(* Logix 5000 project; controller LeakTestAuto vendor 1 type 14 code 226 rev 37.11; software revision 37.01; part 4 of 12 *)
(* tags used below, declared in another part *)
   DateString : String20;
   DateTimeString : String20;
   I_OP220_N3_CONVEYOR_CLEAT : ALIAS FOR Local:3:I.Pt13.Data;
   I_OP220_N3_CONVEYOR_LOAD : ALIAS FOR Local:3:I.Pt12.Data;
   I_OP220_N3_CONVEYOR_UNLOAD : ALIAS FOR Local:3:I.Pt14.Data;
   I_OP220_N3_DUT_PRE_NEST_0 : ALIAS FOR Local:3:I.Pt00.Data;
   I_OP220_N3_DUT_PRE_NEST_1 : ALIAS FOR Local:3:I.Pt01.Data;
   I_OP220_N3_DUT_PRE_NEST_2 : ALIAS FOR Local:3:I.Pt02.Data;
   I_OP220_N3_NEST1_EXTEND : ALIAS FOR Local:3:I.Pt04.Data;
   I_OP220_N3_NEST1_HOME : ALIAS FOR Local:3:I.Pt03.Data;
   I_OP220_N3_NEST2_EXTEND : ALIAS FOR Local:3:I.Pt06.Data;
   I_OP220_N3_NEST2_HOME : ALIAS FOR Local:3:I.Pt05.Data;
   I_OP220_N3_REJECT_BIN_OK : ALIAS FOR Local:3:I.Pt09.Data;
   IOCounterHasRef : BOOL;
   IOTriggerCounts : UDINT[128];
   LastPLCEdit : String20;
   LastPLCEditHistory : String20[20];
   PLC : AOI_PLC;
   ShiftChange : BOOL;
   ShiftNumber : SINT;
   TimeString : String20;
   TON_PLC_BootUp : TIMER;

        [4].Detailed.element_data[2].Variable_code := 13, [4].Detailed.element_data[2].prec_code := 3, [4].Detailed.element_data[2].Unit_code := 12, [4].Detailed.element_data[2].result_measurement := 5.1366444, [4].Detailed.element_data[3].Variable_code := 75, [4].Detailed.element_data[3].prec_code := 2, [4].Detailed.element_data[3].Unit_code := 60, [4].Detailed.element_data[4].Variable_code := 60, [4].Detailed.element_data[4].prec_code := 2, [4].Detailed.element_data[4].Unit_code := 60, [4].Detailed.element_data[4].result_measurement := -0.06984919, [4].Detailed.element_data[5].Variable_code := 56, [4].Detailed.element_data[5].prec_code := 3, [4].Detailed.element_data[5].Unit_code := 41, [4].Detailed.element_data[5].result_measurement := 0.00021420419, [4].Detailed.element_data[6].Variable_code := 55, [4].Detailed.element_data[6].prec_code := 3, [4].Detailed.element_data[6].Unit_code := 12, [4].Detailed.element_data[6].result_measurement := 5.1366444, [4].Detailed.element_data[7].Variable_code := 58, [4].Detailed.element_data[7].prec_code := 2, [4].Detailed.element_data[7].Unit_code := 60, [4].Detailed.element_data[7].result_measurement := -1.0002404, [4].Detailed.element_data[8].Variable_code := 59, [4].Detailed.element_data[8].prec_code := 2, [4].Detailed.element_data[8].Unit_code := 60, [4].Detailed.element_data[8].result_measurement := 1.0002404, [4].Detailed.element_data[9].Variable_code := 12, [4].Detailed.element_data[9].prec_code := 3, [4].Detailed.element_data[9].Unit_code := 12, [4].Detailed.element_data[9].result_measurement := 5.000001, [4].Detailed.element_data[10].Variable_code := 62, [4].Detailed.element_data[10].prec_code := 2, [4].Detailed.element_data[10].Unit_code := 60, [4].Detailed.element_data[10].result_measurement := 1.1002644, [4].Detailed.element_data[11].Variable_code := 21, [4].Detailed.element_data[11].prec_code := 3, [4].Detailed.element_data[11].Unit_code := 41, [4].Detailed.element_data[11].result_measurement := 0.0015180558, [4].Detailed.element_data[12].Variable_code := 25, [4].Detailed.element_data[12].prec_code := 3, [4].Detailed.element_data[12].Unit_code := 41, [4].Detailed.element_data[12].result_measurement := 0.021727756, [4].Detailed.element_data[13].Variable_code := 216, [4].Detailed.element_data[13].prec_code := 3, [4].Detailed.element_data[13].Unit_code := 41, [4].Detailed.element_data[13].result_measurement := 0.00085681677, [4].Detailed.element_data[14].Variable_code := 218, [4].Detailed.element_data[14].prec_code := 3, [4].Detailed.element_data[14].Unit_code := 41, [4].Detailed.element_data[14].result_measurement := 0.01094304, [4].Detailed.element_data[15].Variable_code := 295, [4].Detailed.element_data[15].prec_code := 3, [4].Detailed.element_data[15].Unit_code := 12, [4].Detailed.element_data[15].result_measurement := 5.138372, [5].UID := 41968, [5].Basic.unique_id := 41968, [5].Basic.channel_num := 1, [5].Basic.program_num := 2, [5].Basic.evaluation_code := 1,
        [5].Basic.test_port := 1, [5].Basic.year := 26, [5].Basic.month := 6, [5].Basic.date := 4, [5].Basic.hour := 15, [5].Basic.minute := 9, [5].Basic.second := 31, [5].Basic.flags := 12, [5].Basic.Num_tests := 1, [5].Basic.test_elements.test_type := 66, [5].Basic.test_elements.test_eval := 1, [5].Basic.test_elements.num_elements := 16, [5].Detailed.unique_id := 41968, [5].Detailed.num_elements := 16, [5].Detailed.Test_Type := 66, [5].Detailed.element_data[0].Variable_code := 61, [5].Detailed.element_data[0].prec_code := 2, [5].Detailed.element_data[0].Unit_code := 60, [5].Detailed.element_data[0].result_measurement := -0.054761767, [5].Detailed.element_data[1].Variable_code := 28, [5].Detailed.element_data[1].prec_code := 3, [5].Detailed.element_data[1].Unit_code := 41, [5].Detailed.element_data[1].result_measurement := 0.0005075708, [5].Detailed.element_data[2].Variable_code := 13, [5].Detailed.element_data[2].prec_code := 3, [5].Detailed.element_data[2].Unit_code := 12, [5].Detailed.element_data[2].result_measurement := 5.1372128, [5].Detailed.element_data[3].Variable_code := 75, [5].Detailed.element_data[3].prec_code := 2, [5].Detailed.element_data[3].Unit_code := 60, [5].Detailed.element_data[4].Variable_code := 60, [5].Detailed.element_data[4].prec_code := 2, [5].Detailed.element_data[4].Unit_code := 60, [5].Detailed.element_data[4].result_measurement := -0.05811453, [5].Detailed.element_data[5].Variable_code := 56, [5].Detailed.element_data[5].prec_code := 3, [5].Detailed.element_data[5].Unit_code := 41, [5].Detailed.element_data[5].result_measurement := 0.0003213063, [5].Detailed.element_data[6].Variable_code := 55, [5].Detailed.element_data[6].prec_code := 3, [5].Detailed.element_data[6].Unit_code := 12, [5].Detailed.element_data[6].result_measurement := 5.1372128, [5].Detailed.element_data[7].Variable_code := 58, [5].Detailed.element_data[7].prec_code := 2, [5].Detailed.element_data[7].Unit_code := 60, [5].Detailed.element_data[7].result_measurement := -1.0002404, [5].Detailed.element_data[8].Variable_code := 59, [5].Detailed.element_data[8].prec_code := 2, [5].Detailed.element_data[8].Unit_code := 60, [5].Detailed.element_data[8].result_measurement := 1.0002404, [5].Detailed.element_data[9].Variable_code := 12, [5].Detailed.element_data[9].prec_code := 3, [5].Detailed.element_data[9].Unit_code := 12, [5].Detailed.element_data[9].result_measurement := 5.000001, [5].Detailed.element_data[10].Variable_code := 62, [5].Detailed.element_data[10].prec_code := 2, [5].Detailed.element_data[10].Unit_code := 60, [5].Detailed.element_data[10].result_measurement := 1.1002644, [5].Detailed.element_data[11].Variable_code := 21, [5].Detailed.element_data[11].prec_code := 3,
        [5].Detailed.element_data[11].Unit_code := 41, [5].Detailed.element_data[11].result_measurement := 0.0015180558, [5].Detailed.element_data[12].Variable_code := 25, [5].Detailed.element_data[12].prec_code := 3, [5].Detailed.element_data[12].Unit_code := 41, [5].Detailed.element_data[12].result_measurement := 0.021727756, [5].Detailed.element_data[13].Variable_code := 216, [5].Detailed.element_data[13].prec_code := 3, [5].Detailed.element_data[13].Unit_code := 41, [5].Detailed.element_data[13].result_measurement := 0.00085681677, [5].Detailed.element_data[14].Variable_code := 218, [5].Detailed.element_data[14].prec_code := 3, [5].Detailed.element_data[14].Unit_code := 41, [5].Detailed.element_data[14].result_measurement := 0.01094304, [5].Detailed.element_data[15].Variable_code := 295, [5].Detailed.element_data[15].prec_code := 3, [5].Detailed.element_data[15].Unit_code := 12, [5].Detailed.element_data[15].result_measurement := 5.139271, [6].UID := 42010, [6].Basic.unique_id := 42010, [6].Basic.channel_num := 1, [6].Basic.program_num := 2, [6].Basic.evaluation_code := 1, [6].Basic.test_port := 1, [6].Basic.year := 26, [6].Basic.month := 6, [6].Basic.date := 5, [6].Basic.hour := 10, [6].Basic.minute := 13, [6].Basic.second := 42, [6].Basic.flags := 12, [6].Basic.Num_tests := 1, [6].Basic.test_elements.test_type := 66, [6].Basic.test_elements.test_eval := 1, [6].Basic.test_elements.num_elements := 16, [6].Detailed.unique_id := 42010, [6].Detailed.num_elements := 16, [6].Detailed.Test_Type := 66, [6].Detailed.element_data[0].Variable_code := 61, [6].Detailed.element_data[0].prec_code := 2, [6].Detailed.element_data[0].Unit_code := 60, [6].Detailed.element_data[0].result_measurement := -0.067055225, [6].Detailed.element_data[1].Variable_code := 28, [6].Detailed.element_data[1].prec_code := 3, [6].Detailed.element_data[1].Unit_code := 41, [6].Detailed.element_data[1].result_measurement := 0.00027939677, [6].Detailed.element_data[2].Variable_code := 13, [6].Detailed.element_data[2].prec_code := 3, [6].Detailed.element_data[2].Unit_code := 12, [6].Detailed.element_data[2].result_measurement := 5.1023254, [6].Detailed.element_data[3].Variable_code := 75, [6].Detailed.element_data[3].prec_code := 2, [6].Detailed.element_data[3].Unit_code := 60, [6].Detailed.element_data[4].Variable_code := 60, [6].Detailed.element_data[4].prec_code := 2, [6].Detailed.element_data[4].Unit_code := 60, [6].Detailed.element_data[4].result_measurement := -0.07208437, [6].Detailed.element_data[5].Variable_code := 56, [6].Detailed.element_data[5].prec_code := 3, [6].Detailed.element_data[5].Unit_code := 41,
        [6].Detailed.element_data[5].result_measurement := 0.00019092113, [6].Detailed.element_data[6].Variable_code := 55, [6].Detailed.element_data[6].prec_code := 3, [6].Detailed.element_data[6].Unit_code := 12, [6].Detailed.element_data[6].result_measurement := 5.1023254, [6].Detailed.element_data[7].Variable_code := 58, [6].Detailed.element_data[7].prec_code := 2, [6].Detailed.element_data[7].Unit_code := 60, [6].Detailed.element_data[7].result_measurement := -1.0002404, [6].Detailed.element_data[8].Variable_code := 59, [6].Detailed.element_data[8].prec_code := 2, [6].Detailed.element_data[8].Unit_code := 60, [6].Detailed.element_data[8].result_measurement := 1.0002404, [6].Detailed.element_data[9].Variable_code := 12, [6].Detailed.element_data[9].prec_code := 3, [6].Detailed.element_data[9].Unit_code := 12, [6].Detailed.element_data[9].result_measurement := 5.000001, [6].Detailed.element_data[10].Variable_code := 62, [6].Detailed.element_data[10].prec_code := 2, [6].Detailed.element_data[10].Unit_code := 60, [6].Detailed.element_data[10].result_measurement := 1.1002644, [6].Detailed.element_data[11].Variable_code := 21, [6].Detailed.element_data[11].prec_code := 3, [6].Detailed.element_data[11].Unit_code := 41, [6].Detailed.element_data[11].result_measurement := 0.0015180558, [6].Detailed.element_data[12].Variable_code := 25, [6].Detailed.element_data[12].prec_code := 3, [6].Detailed.element_data[12].Unit_code := 41, [6].Detailed.element_data[12].result_measurement := 0.021727756, [6].Detailed.element_data[13].Variable_code := 216, [6].Detailed.element_data[13].prec_code := 3, [6].Detailed.element_data[13].Unit_code := 41, [6].Detailed.element_data[13].result_measurement := 0.00085681677, [6].Detailed.element_data[14].Variable_code := 218, [6].Detailed.element_data[14].prec_code := 3, [6].Detailed.element_data[14].Unit_code := 41, [6].Detailed.element_data[14].result_measurement := 0.01094304, [6].Detailed.element_data[15].Variable_code := 295, [6].Detailed.element_data[15].prec_code := 3, [6].Detailed.element_data[15].Unit_code := 12, [6].Detailed.element_data[15].result_measurement := 5.1039925, [7].UID := 42013, [7].Basic.unique_id := 42013, [7].Basic.channel_num := 1, [7].Basic.program_num := 2, [7].Basic.evaluation_code := 1, [7].Basic.test_port := 1, [7].Basic.year := 26, [7].Basic.month := 6, [7].Basic.date := 5, [7].Basic.hour := 10, [7].Basic.minute := 17, [7].Basic.second := 34, [7].Basic.flags := 12, [7].Basic.Num_tests := 1, [7].Basic.test_elements.test_type := 66, [7].Basic.test_elements.test_eval := 1, [7].Basic.test_elements.num_elements := 16, [7].Detailed.unique_id := 42013, [7].Detailed.num_elements := 16,
        [7].Detailed.Test_Type := 66, [7].Detailed.element_data[0].Variable_code := 61, [7].Detailed.element_data[0].prec_code := 2, [7].Detailed.element_data[0].Unit_code := 60, [7].Detailed.element_data[0].result_measurement := -0.07040799, [7].Detailed.element_data[1].Variable_code := 28, [7].Detailed.element_data[1].prec_code := 3, [7].Detailed.element_data[1].Unit_code := 41, [7].Detailed.element_data[1].result_measurement := 0.00022351742, [7].Detailed.element_data[2].Variable_code := 13, [7].Detailed.element_data[2].prec_code := 3, [7].Detailed.element_data[2].Unit_code := 12, [7].Detailed.element_data[2].result_measurement := 5.101585, [7].Detailed.element_data[3].Variable_code := 75, [7].Detailed.element_data[3].prec_code := 2, [7].Detailed.element_data[3].Unit_code := 60, [7].Detailed.element_data[4].Variable_code := 60, [7].Detailed.element_data[4].prec_code := 2, [7].Detailed.element_data[4].Unit_code := 60, [7].Detailed.element_data[4].result_measurement := -0.07711351, [7].Detailed.element_data[5].Variable_code := 56, [7].Detailed.element_data[5].prec_code := 3, [7].Detailed.element_data[5].Unit_code := 41, [7].Detailed.element_data[5].result_measurement := 0.00014901161, [7].Detailed.element_data[6].Variable_code := 55, [7].Detailed.element_data[6].prec_code := 3, [7].Detailed.element_data[6].Unit_code := 12, [7].Detailed.element_data[6].result_measurement := 5.101585, [7].Detailed.element_data[7].Variable_code := 58, [7].Detailed.element_data[7].prec_code := 2, [7].Detailed.element_data[7].Unit_code := 60, [7].Detailed.element_data[7].result_measurement := -1.0002404, [7].Detailed.element_data[8].Variable_code := 59, [7].Detailed.element_data[8].prec_code := 2, [7].Detailed.element_data[8].Unit_code := 60, [7].Detailed.element_data[8].result_measurement := 1.0002404, [7].Detailed.element_data[9].Variable_code := 12, [7].Detailed.element_data[9].prec_code := 3, [7].Detailed.element_data[9].Unit_code := 12, [7].Detailed.element_data[9].result_measurement := 5.000001, [7].Detailed.element_data[10].Variable_code := 62, [7].Detailed.element_data[10].prec_code := 2, [7].Detailed.element_data[10].Unit_code := 60, [7].Detailed.element_data[10].result_measurement := 1.1002644, [7].Detailed.element_data[11].Variable_code := 21, [7].Detailed.element_data[11].prec_code := 3, [7].Detailed.element_data[11].Unit_code := 41, [7].Detailed.element_data[11].result_measurement := 0.0015180558, [7].Detailed.element_data[12].Variable_code := 25, [7].Detailed.element_data[12].prec_code := 3, [7].Detailed.element_data[12].Unit_code := 41, [7].Detailed.element_data[12].result_measurement := 0.021727756, [7].Detailed.element_data[13].Variable_code := 216, [7].Detailed.element_data[13].prec_code := 3, [7].Detailed.element_data[13].Unit_code := 41, [7].Detailed.element_data[13].result_measurement := 0.00085681677, [7].Detailed.element_data[14].Variable_code := 218, [7].Detailed.element_data[14].prec_code := 3, [7].Detailed.element_data[14].Unit_code := 41, [7].Detailed.element_data[14].result_measurement := 0.01094304,
        [7].Detailed.element_data[15].Variable_code := 295, [7].Detailed.element_data[15].prec_code := 3, [7].Detailed.element_data[15].Unit_code := 12, [7].Detailed.element_data[15].result_measurement := 5.103038, [8].UID := 42016, [8].Basic.unique_id := 42016, [8].Basic.channel_num := 1, [8].Basic.program_num := 2, [8].Basic.evaluation_code := 1, [8].Basic.test_port := 1, [8].Basic.year := 26, [8].Basic.month := 6, [8].Basic.date := 5, [8].Basic.hour := 10, [8].Basic.minute := 18, [8].Basic.second := 33, [8].Basic.flags := 12, [8].Basic.Num_tests := 1, [8].Basic.test_elements.test_type := 66, [8].Basic.test_elements.test_eval := 1, [8].Basic.test_elements.num_elements := 16, [8].Detailed.unique_id := 42016, [8].Detailed.num_elements := 16, [8].Detailed.Test_Type := 66, [8].Detailed.element_data[0].Variable_code := 61, [8].Detailed.element_data[0].prec_code := 2, [8].Detailed.element_data[0].Unit_code := 60, [8].Detailed.element_data[0].result_measurement := -0.0692904, [8].Detailed.element_data[1].Variable_code := 28, [8].Detailed.element_data[1].prec_code := 3, [8].Detailed.element_data[1].Unit_code := 41, [8].Detailed.element_data[1].result_measurement := 0.00023748726, [8].Detailed.element_data[2].Variable_code := 13, [8].Detailed.element_data[2].prec_code := 3, [8].Detailed.element_data[2].Unit_code := 12, [8].Detailed.element_data[2].result_measurement := 5.1036057, [8].Detailed.element_data[3].Variable_code := 75, [8].Detailed.element_data[3].prec_code := 2, [8].Detailed.element_data[3].Unit_code := 60, [8].Detailed.element_data[4].Variable_code := 60, [8].Detailed.element_data[4].prec_code := 2, [8].Detailed.element_data[4].Unit_code := 60, [8].Detailed.element_data[4].result_measurement := -0.073201954, [8].Detailed.element_data[5].Variable_code := 56, [8].Detailed.element_data[5].prec_code := 3, [8].Detailed.element_data[5].Unit_code := 41, [8].Detailed.element_data[5].result_measurement := 0.0001816079, [8].Detailed.element_data[6].Variable_code := 55, [8].Detailed.element_data[6].prec_code := 3, [8].Detailed.element_data[6].Unit_code := 12, [8].Detailed.element_data[6].result_measurement := 5.1036057, [8].Detailed.element_data[7].Variable_code := 58, [8].Detailed.element_data[7].prec_code := 2, [8].Detailed.element_data[7].Unit_code := 60, [8].Detailed.element_data[7].result_measurement := -1.0002404, [8].Detailed.element_data[8].Variable_code := 59, [8].Detailed.element_data[8].prec_code := 2, [8].Detailed.element_data[8].Unit_code := 60, [8].Detailed.element_data[8].result_measurement := 1.0002404, [8].Detailed.element_data[9].Variable_code := 12,
        [8].Detailed.element_data[9].prec_code := 3, [8].Detailed.element_data[9].Unit_code := 12, [8].Detailed.element_data[9].result_measurement := 5.000001, [8].Detailed.element_data[10].Variable_code := 62, [8].Detailed.element_data[10].prec_code := 2, [8].Detailed.element_data[10].Unit_code := 60, [8].Detailed.element_data[10].result_measurement := 1.1002644, [8].Detailed.element_data[11].Variable_code := 21, [8].Detailed.element_data[11].prec_code := 3, [8].Detailed.element_data[11].Unit_code := 41, [8].Detailed.element_data[11].result_measurement := 0.0015180558, [8].Detailed.element_data[12].Variable_code := 25, [8].Detailed.element_data[12].prec_code := 3, [8].Detailed.element_data[12].Unit_code := 41, [8].Detailed.element_data[12].result_measurement := 0.021727756, [8].Detailed.element_data[13].Variable_code := 216, [8].Detailed.element_data[13].prec_code := 3, [8].Detailed.element_data[13].Unit_code := 41, [8].Detailed.element_data[13].result_measurement := 0.00085681677, [8].Detailed.element_data[14].Variable_code := 218, [8].Detailed.element_data[14].prec_code := 3, [8].Detailed.element_data[14].Unit_code := 41, [8].Detailed.element_data[14].result_measurement := 0.01094304, [8].Detailed.element_data[15].Variable_code := 295, [8].Detailed.element_data[15].prec_code := 3, [8].Detailed.element_data[15].Unit_code := 12, [8].Detailed.element_data[15].result_measurement := 5.1049933);
   CTS2_ResultHistoryVol : udt_CTS_RESULT[10] := ([0].UID := 41958, [0].Basic.unique_id := 41958, [0].Basic.channel_num := 1, [0].Basic.program_num := 1, [0].Basic.evaluation_code := 1, [0].Basic.test_port := 1, [0].Basic.year := 26, [0].Basic.month := 6, [0].Basic.date := 4, [0].Basic.hour := 15, [0].Basic.minute := 3, [0].Basic.second := 10, [0].Basic.flags := 12, [0].Basic.Num_tests := 1, [0].Basic.test_elements.test_type := 69, [0].Basic.test_elements.test_eval := 1, [0].Basic.test_elements.num_elements := 4, [0].Detailed.unique_id := 41958, [0].Detailed.num_elements := 4, [0].Detailed.Test_Type := 69, [0].Detailed.element_data[0].Variable_code := 245, [0].Detailed.element_data[0].prec_code := 2, [0].Detailed.element_data[0].Unit_code := 165, [0].Detailed.element_data[0].result_measurement := 186.90665, [0].Detailed.element_data[1].Variable_code := 13, [0].Detailed.element_data[1].prec_code := 3, [0].Detailed.element_data[1].Unit_code := 12, [0].Detailed.element_data[1].result_measurement := 1.7801206, [0].Detailed.element_data[2].Variable_code := 247, [0].Detailed.element_data[2].prec_code := 3, [0].Detailed.element_data[2].Unit_code := 12, [0].Detailed.element_data[2].result_measurement := 5.1072845, [0].Detailed.element_data[3].Variable_code := 295, [0].Detailed.element_data[3].prec_code := 3, [0].Detailed.element_data[3].Unit_code := 12, [0].Detailed.element_data[3].result_measurement := 5.1086583, [1].UID := 41961, [1].Basic.unique_id := 41961, [1].Basic.channel_num := 1, [1].Basic.program_num := 1, [1].Basic.evaluation_code := 1, [1].Basic.test_port := 1, [1].Basic.year := 26, [1].Basic.month := 6, [1].Basic.date := 4, [1].Basic.hour := 15, [1].Basic.minute := 6, [1].Basic.second := 33, [1].Basic.flags := 12, [1].Basic.Num_tests := 1, [1].Basic.test_elements.test_type := 69, [1].Basic.test_elements.test_eval := 1, [1].Basic.test_elements.num_elements := 4, [1].Detailed.unique_id := 41961, [1].Detailed.num_elements := 4, [1].Detailed.Test_Type := 69, [1].Detailed.element_data[0].Variable_code := 245, [1].Detailed.element_data[0].prec_code := 2, [1].Detailed.element_data[0].Unit_code := 165, [1].Detailed.element_data[0].result_measurement := 186.6259,
        [1].Detailed.element_data[1].Variable_code := 13, [1].Detailed.element_data[1].prec_code := 3, [1].Detailed.element_data[1].Unit_code := 12, [1].Detailed.element_data[1].result_measurement := 1.7820624, [1].Detailed.element_data[2].Variable_code := 247, [1].Detailed.element_data[2].prec_code := 3, [1].Detailed.element_data[2].Unit_code := 12, [1].Detailed.element_data[2].result_measurement := 5.1078525, [1].Detailed.element_data[3].Variable_code := 295, [1].Detailed.element_data[3].prec_code := 3, [1].Detailed.element_data[3].Unit_code := 12, [1].Detailed.element_data[3].result_measurement := 5.1083417, [2].UID := 41964, [2].Basic.unique_id := 41964, [2].Basic.channel_num := 1, [2].Basic.program_num := 1, [2].Basic.evaluation_code := 1, [2].Basic.test_port := 1, [2].Basic.year := 26, [2].Basic.month := 6, [2].Basic.date := 4, [2].Basic.hour := 15, [2].Basic.minute := 7, [2].Basic.second := 46, [2].Basic.flags := 12, [2].Basic.Num_tests := 1, [2].Basic.test_elements.test_type := 69, [2].Basic.test_elements.test_eval := 1, [2].Basic.test_elements.num_elements := 4, [2].Detailed.unique_id := 41964, [2].Detailed.num_elements := 4, [2].Detailed.Test_Type := 69, [2].Detailed.element_data[0].Variable_code := 245, [2].Detailed.element_data[0].prec_code := 2, [2].Detailed.element_data[0].Unit_code := 165, [2].Detailed.element_data[0].result_measurement := 186.70047, [2].Detailed.element_data[1].Variable_code := 13, [2].Detailed.element_data[1].prec_code := 3, [2].Detailed.element_data[1].Unit_code := 12, [2].Detailed.element_data[1].result_measurement := 1.7814804, [2].Detailed.element_data[2].Variable_code := 247, [2].Detailed.element_data[2].prec_code := 3, [2].Detailed.element_data[2].Unit_code := 12, [2].Detailed.element_data[2].result_measurement := 5.1075125, [2].Detailed.element_data[3].Variable_code := 295, [2].Detailed.element_data[3].prec_code := 3, [2].Detailed.element_data[3].Unit_code := 12, [2].Detailed.element_data[3].result_measurement := 5.1079783, [3].UID := 41967, [3].Basic.unique_id := 41967, [3].Basic.channel_num := 1, [3].Basic.program_num := 1, [3].Basic.evaluation_code := 1, [3].Basic.test_port := 1, [3].Basic.year := 26, [3].Basic.month := 6, [3].Basic.date := 4, [3].Basic.hour := 15, [3].Basic.minute := 9, [3].Basic.second := 24,
        [3].Basic.flags := 12, [3].Basic.Num_tests := 1, [3].Basic.test_elements.test_type := 69, [3].Basic.test_elements.test_eval := 1, [3].Basic.test_elements.num_elements := 4, [3].Detailed.unique_id := 41967, [3].Detailed.num_elements := 4, [3].Detailed.Test_Type := 69, [3].Detailed.element_data[0].Variable_code := 245, [3].Detailed.element_data[0].prec_code := 2, [3].Detailed.element_data[0].Unit_code := 165, [3].Detailed.element_data[0].result_measurement := 186.79054, [3].Detailed.element_data[1].Variable_code := 13, [3].Detailed.element_data[1].prec_code := 3, [3].Detailed.element_data[1].Unit_code := 12, [3].Detailed.element_data[1].result_measurement := 1.7802324, [3].Detailed.element_data[2].Variable_code := 247, [3].Detailed.element_data[2].prec_code := 3, [3].Detailed.element_data[2].Unit_code := 12, [3].Detailed.element_data[2].result_measurement := 5.1055384, [3].Detailed.element_data[3].Variable_code := 295, [3].Detailed.element_data[3].prec_code := 3, [3].Detailed.element_data[3].Unit_code := 12, [3].Detailed.element_data[3].result_measurement := 5.1066375, [4].UID := 42009, [4].Basic.unique_id := 42009, [4].Basic.channel_num := 1, [4].Basic.program_num := 1, [4].Basic.evaluation_code := 1, [4].Basic.test_port := 1, [4].Basic.year := 26, [4].Basic.month := 6, [4].Basic.date := 5, [4].Basic.hour := 10, [4].Basic.minute := 13, [4].Basic.second := 35, [4].Basic.flags := 12, [4].Basic.Num_tests := 1, [4].Basic.test_elements.test_type := 69, [4].Basic.test_elements.test_eval := 1, [4].Basic.test_elements.num_elements := 4, [4].Detailed.unique_id := 42009, [4].Detailed.num_elements := 4, [4].Detailed.Test_Type := 69, [4].Detailed.element_data[0].Variable_code := 245, [4].Detailed.element_data[0].prec_code := 2, [4].Detailed.element_data[0].Unit_code := 165, [4].Detailed.element_data[0].result_measurement := 185.74803, [4].Detailed.element_data[1].Variable_code := 13, [4].Detailed.element_data[1].prec_code := 3, [4].Detailed.element_data[1].Unit_code := 12, [4].Detailed.element_data[1].result_measurement := 1.7781556, [4].Detailed.element_data[2].Variable_code := 247, [4].Detailed.element_data[2].prec_code := 3, [4].Detailed.element_data[2].Unit_code := 12, [4].Detailed.element_data[2].result_measurement := 5.0810447, [4].Detailed.element_data[3].Variable_code := 295, [4].Detailed.element_data[3].prec_code := 3, [4].Detailed.element_data[3].Unit_code := 12, [4].Detailed.element_data[3].result_measurement := 5.081105,
        [5].UID := 42012, [5].Basic.unique_id := 42012, [5].Basic.channel_num := 1, [5].Basic.program_num := 1, [5].Basic.evaluation_code := 1, [5].Basic.test_port := 1, [5].Basic.year := 26, [5].Basic.month := 6, [5].Basic.date := 5, [5].Basic.hour := 10, [5].Basic.minute := 17, [5].Basic.second := 27, [5].Basic.flags := 12, [5].Basic.Num_tests := 1, [5].Basic.test_elements.test_type := 69, [5].Basic.test_elements.test_eval := 1, [5].Basic.test_elements.num_elements := 4, [5].Detailed.unique_id := 42012, [5].Detailed.num_elements := 4, [5].Detailed.Test_Type := 69, [5].Detailed.element_data[0].Variable_code := 245, [5].Detailed.element_data[0].prec_code := 2, [5].Detailed.element_data[0].Unit_code := 165, [5].Detailed.element_data[0].result_measurement := 185.72876, [5].Detailed.element_data[1].Variable_code := 13, [5].Detailed.element_data[1].prec_code := 3, [5].Detailed.element_data[1].Unit_code := 12, [5].Detailed.element_data[1].result_measurement := 1.7785281, [5].Detailed.element_data[2].Variable_code := 247, [5].Detailed.element_data[2].prec_code := 3, [5].Detailed.element_data[2].Unit_code := 12, [5].Detailed.element_data[2].result_measurement := 5.081766, [5].Detailed.element_data[3].Variable_code := 295, [5].Detailed.element_data[3].prec_code := 3, [5].Detailed.element_data[3].Unit_code := 12, [5].Detailed.element_data[3].result_measurement := 5.0830374, [6].UID := 42015, [6].Basic.unique_id := 42015, [6].Basic.channel_num := 1, [6].Basic.program_num := 1, [6].Basic.evaluation_code := 1, [6].Basic.test_port := 1, [6].Basic.year := 26, [6].Basic.month := 6, [6].Basic.date := 5, [6].Basic.hour := 10, [6].Basic.minute := 18, [6].Basic.second := 26, [6].Basic.flags := 12, [6].Basic.Num_tests := 1, [6].Basic.test_elements.test_type := 69, [6].Basic.test_elements.test_eval := 1, [6].Basic.test_elements.num_elements := 4, [6].Detailed.unique_id := 42015, [6].Detailed.num_elements := 4, [6].Detailed.Test_Type := 69, [6].Detailed.element_data[0].Variable_code := 245, [6].Detailed.element_data[0].prec_code := 2, [6].Detailed.element_data[0].Unit_code := 165, [6].Detailed.element_data[0].result_measurement := 185.95625,
        [6].Detailed.element_data[1].Variable_code := 13, [6].Detailed.element_data[1].prec_code := 3, [6].Detailed.element_data[1].Unit_code := 12, [6].Detailed.element_data[1].result_measurement := 1.778258, [6].Detailed.element_data[2].Variable_code := 247, [6].Detailed.element_data[2].prec_code := 3, [6].Detailed.element_data[2].Unit_code := 12, [6].Detailed.element_data[2].result_measurement := 5.08504, [6].Detailed.element_data[3].Variable_code := 295, [6].Detailed.element_data[3].prec_code := 3, [6].Detailed.element_data[3].Unit_code := 12, [6].Detailed.element_data[3].result_measurement := 5.086218, [7].UID := 42018, [7].Basic.unique_id := 42018, [7].Basic.channel_num := 1, [7].Basic.program_num := 1, [7].Basic.evaluation_code := 2, [7].Basic.test_port := 1, [7].Basic.year := 26, [7].Basic.month := 6, [7].Basic.date := 5, [7].Basic.hour := 10, [7].Basic.minute := 54, [7].Basic.second := 14, [7].Basic.flags := 12, [7].Basic.Num_tests := 1, [7].Basic.test_elements.test_type := 69, [7].Basic.test_elements.test_eval := 2, [7].Basic.test_elements.num_elements := 4, [7].Detailed.unique_id := 42018, [7].Detailed.num_elements := 4, [7].Detailed.Test_Type := 69, [7].Detailed.element_data[0].Variable_code := 245, [7].Detailed.element_data[0].prec_code := 2, [7].Detailed.element_data[0].Unit_code := 165, [7].Detailed.element_data[0].result_measurement := 1000.0, [7].Detailed.element_data[1].Variable_code := 13, [7].Detailed.element_data[1].prec_code := 3, [7].Detailed.element_data[1].Unit_code := 12, [7].Detailed.element_data[1].result_measurement := 0.0002933666, [7].Detailed.element_data[2].Variable_code := 247, [7].Detailed.element_data[2].prec_code := 3, [7].Detailed.element_data[2].Unit_code := 12, [7].Detailed.element_data[2].result_measurement := 5.0650864, [7].Detailed.element_data[3].Variable_code := 295, [7].Detailed.element_data[3].prec_code := 3, [7].Detailed.element_data[3].Unit_code := 12, [7].Detailed.element_data[3].result_measurement := 5.0667486, [8].UID := 42020, [8].Basic.unique_id := 42020, [8].Basic.channel_num := 1, [8].Basic.program_num := 1, [8].Basic.evaluation_code := 1, [8].Basic.test_port := 1, [8].Basic.year := 26, [8].Basic.month := 6, [8].Basic.date := 5, [8].Basic.hour := 10, [8].Basic.minute := 54, [8].Basic.second := 35,
        [8].Basic.flags := 12, [8].Basic.Num_tests := 1, [8].Basic.test_elements.test_type := 69, [8].Basic.test_elements.test_eval := 1, [8].Basic.test_elements.num_elements := 4, [8].Detailed.unique_id := 42020, [8].Detailed.num_elements := 4, [8].Detailed.Test_Type := 69, [8].Detailed.element_data[0].Variable_code := 245, [8].Detailed.element_data[0].prec_code := 2, [8].Detailed.element_data[0].Unit_code := 165, [8].Detailed.element_data[0].result_measurement := 186.5566, [8].Detailed.element_data[1].Variable_code := 13, [8].Detailed.element_data[1].prec_code := 3, [8].Detailed.element_data[1].Unit_code := 12, [8].Detailed.element_data[1].result_measurement := 1.768372, [8].Detailed.element_data[2].Variable_code := 247, [8].Detailed.element_data[2].prec_code := 3, [8].Detailed.element_data[2].Unit_code := 12, [8].Detailed.element_data[2].result_measurement := 5.0673866, [8].Detailed.element_data[3].Variable_code := 295, [8].Detailed.element_data[3].prec_code := 3, [8].Detailed.element_data[3].Unit_code := 12, [8].Detailed.element_data[3].result_measurement := 5.068574, [9].UID := 42023, [9].Basic.unique_id := 42023, [9].Basic.channel_num := 1, [9].Basic.program_num := 1, [9].Basic.evaluation_code := 1, [9].Basic.test_port := 1, [9].Basic.year := 26, [9].Basic.month := 6, [9].Basic.date := 5, [9].Basic.hour := 10, [9].Basic.minute := 55, [9].Basic.second := 43, [9].Basic.flags := 12, [9].Basic.Num_tests := 1, [9].Basic.test_elements.test_type := 69, [9].Basic.test_elements.test_eval := 1, [9].Basic.test_elements.num_elements := 4, [9].Detailed.unique_id := 42023, [9].Detailed.num_elements := 4, [9].Detailed.Test_Type := 69, [9].Detailed.element_data[0].Variable_code := 245, [9].Detailed.element_data[0].prec_code := 2, [9].Detailed.element_data[0].Unit_code := 165, [9].Detailed.element_data[0].result_measurement := 186.64526, [9].Detailed.element_data[1].Variable_code := 13, [9].Detailed.element_data[1].prec_code := 3, [9].Detailed.element_data[1].Unit_code := 12, [9].Detailed.element_data[1].result_measurement := 1.7689215, [9].Detailed.element_data[2].Variable_code := 247, [9].Detailed.element_data[2].prec_code := 3, [9].Detailed.element_data[2].Unit_code := 12, [9].Detailed.element_data[2].result_measurement := 5.07053, [9].Detailed.element_data[3].Variable_code := 295, [9].Detailed.element_data[3].prec_code := 3, [9].Detailed.element_data[3].Unit_code := 12, [9].Detailed.element_data[3].result_measurement := 5.0715685);
   CTS2_Seq : udt_SequenceStructure_X64 := (CycleDone := 1, CurrentStep := 9000, NextStep := 9000, ONS := -32767, StepHistory[0] := 1000, StepHistory[1] := 1010, StepHistory[2] := 1020, StepHistory[3] := 1030, StepHistory[4] := 2000, StepHistory[5] := 2010, StepHistory[6] := 2020, StepHistory[7] := 2030, StepHistory[8] := 2000, StepHistory[9] := 2010, StepHistory[10] := 2020, StepHistory[11] := 2030, StepHistory[12] := 9000, StepHistory[13] := 1000, StepHistory[14] := 1010, StepHistory[15] := 1020, StepHistory[16] := 1030, StepHistory[17] := 2000, StepHistory[18] := 2010, StepHistory[19] := 2020, StepHistory[20] := 2030, StepHistory[21] := 2000, StepHistory[22] := 2010, StepHistory[23] := 2020, StepHistory[24] := 2030, StepHistory[25] := 9000, StepHistory[26] := 1000, StepHistory[27] := 1010, StepHistory[28] := 1020, StepHistory[29] := 1030, StepHistory[30] := 2000, StepHistory[31] := 2010, StepHistory[32] := 2020, StepHistory[33] := 2030, StepHistory[34] := 9000, StepHistory[35] := 1000, StepHistory[36] := 1010, StepHistory[37] := 1020, StepHistory[38] := 1030, StepHistory[39] := 2000, StepHistory[40] := 2010, StepHistory[41] := 2020, StepHistory[42] := 2030, StepHistory[43] := 2000, StepHistory[44] := 2010, StepHistory[45] := 2020, StepHistory[46] := 2030, StepHistory[47] := 9000, StepHistory[48] := 1000, StepHistory[49] := 1010, StepHistory[50] := 1020, StepHistory[51] := 1030, StepHistory[52] := 2000, StepHistory[53] := 2010, StepHistory[54] := 2020, StepHistory[55] := 2030,
        StepHistory[56] := 2000, StepHistory[57] := 2010, StepHistory[58] := 2020, StepHistory[59] := 2030, StepHistory[60] := 9000, StepHistory[61] := 1000, StepHistory[62] := 1010, StepHistory[63] := 1020, AverageCycleTime := 1.0542, CycleTimeHistory[0] := 2.209, CycleTimeHistory[1] := 2.209, CycleTimeHistory[3] := 1.206, CycleTimeHistory[4] := 2.209, CycleTimeHistory[5] := 2.209, CycleTimeHistory[8] := 0.5, StepTimeHistory[1] := 0.199, StepTimeHistory[2] := 0.199, StepTimeHistory[3] := 0.199, StepTimeHistory[5] := 1.0, StepTimeHistory[6] := 1.0, StepTimeHistory[7] := 1.0, StepTimeHistory[9] := 0.999, StepTimeHistory[10] := 0.999, StepTimeHistory[11] := 0.999, StepTimeHistory[12] := 0.999, StepTimeHistory[14] := 0.199, StepTimeHistory[15] := 0.199, StepTimeHistory[16] := 0.199, StepTimeHistory[18] := 1.0, StepTimeHistory[19] := 1.0, StepTimeHistory[20] := 1.0, StepTimeHistory[22] := 0.999, StepTimeHistory[23] := 0.999, StepTimeHistory[24] := 0.999, StepTimeHistory[27] := 0.199, StepTimeHistory[28] := 0.199, StepTimeHistory[29] := 0.199, StepTimeHistory[31] := 1.0, StepTimeHistory[32] := 1.0, StepTimeHistory[33] := 1.0, StepTimeHistory[34] := 1.0, StepTimeHistory[36] := 0.199, StepTimeHistory[37] := 0.199, StepTimeHistory[38] := 0.199, StepTimeHistory[40] := 0.999, StepTimeHistory[41] := 0.999, StepTimeHistory[42] := 0.999, StepTimeHistory[44] := 1.0, StepTimeHistory[45] := 1.0, StepTimeHistory[46] := 1.0, StepTimeHistory[47] := 1.0, StepTimeHistory[49] := 0.2, StepTimeHistory[50] := 0.2, StepTimeHistory[51] := 0.2, StepTimeHistory[53] := 0.999, StepTimeHistory[54] := 0.999, StepTimeHistory[55] := 0.999, StepTimeHistory[57] := 0.999, StepTimeHistory[58] := 0.999, StepTimeHistory[59] := 0.999,
        StepTimeHistory[62] := 0.199, StepTimeHistory[63] := 0.299, StepTimer.PRE := 999999999, CycleTimer.PRE := 999999999);
   CTS2_SeqUID : DINT := 42054;
   CTS2_UIDMsg : MESSAGE;
        MessageParameters(ServiceCode := 16#0010, LocalElement := CTS2_Result.UID, ...)
   CTS2_WriteMsg : MESSAGE;
        MessageParameters(ServiceCode := 16#0010, LocalElement := CTS2_BarcodeWrite.DATA[0], ...)
   CTS_NoResult : udt_CTS_RESULT;
   CTS_ResultDump : udt_CTS_RESULT := (UID := 41955, Basic.unique_id := 41955, Basic.channel_num := 1, Basic.program_num := 1, Basic.evaluation_code := 1, Basic.test_port := 1, Basic.year := 26, Basic.month := 6, Basic.date := 4, Basic.hour := 14, Basic.minute := 58, Basic.second := 18, Basic.flags := 12, Basic.Num_tests := 1, Basic.test_elements.test_type := 69, Basic.test_elements.test_eval := 1, Basic.test_elements.num_elements := 4, Detailed.unique_id := 41955, Detailed.num_elements := 4, Detailed.Test_Type := 69, Detailed.element_data[0].Variable_code := 245, Detailed.element_data[0].prec_code := 2, Detailed.element_data[0].Unit_code := 165, Detailed.element_data[0].result_measurement := 186.52744, Detailed.element_data[1].Variable_code := 13, Detailed.element_data[1].prec_code := 3, Detailed.element_data[1].Unit_code := 12, Detailed.element_data[1].result_measurement := 1.782449, Detailed.element_data[2].Variable_code := 247, Detailed.element_data[2].prec_code := 3, Detailed.element_data[2].Unit_code := 12, Detailed.element_data[2].result_measurement := 5.1072054, Detailed.element_data[3].Variable_code := 295, Detailed.element_data[3].prec_code := 3, Detailed.element_data[3].Unit_code := 12, Detailed.element_data[3].result_measurement := 5.109105);
   CurrentDUTData : udt_DUTHistory[2] := ([0].Barcode := 'B252620969', [1].Barcode := 'B252620970');
   DryCycle_N1Ready : BOOL;
   DryCycle_N2Ready : BOOL;
   DUTHistoryDump : udt_DUTHistory := (Barcode := 'A252620388');
   DUTTestHistory : udt_DUTHistory[10] := ([0].Barcode := 'A252620388', [1].Barcode := 'A252620388', [2].Barcode := 'A252620388', [3].Barcode := 'A252620388', [4].Barcode := 'A252620388', [5].Barcode := 'A252620388', [6].Barcode := 'A252620388', [7].Barcode := 'A252620388', [8].Barcode := 'A252620388', [9].Barcode := 'A252620388');
   EIPTemplateCommStatus : AOI_CommStatus;
   EIPTemplateDeviceInput : udt_EIPTemplateData;
   EIPTemplateDeviceOutput : udt_EIPTemplateData;
   EIPTemplateLocalInput : udt_EIPTemplateLocalInput;
   EIPTemplateLocalOutput : udt_EIPTemplateLocalOutput;
   FailCount : COUNTER := (PRE := 10);
   FaultsAndWarnings : STRING[96] := ([0] := 'Main power off', [1] := 'Main air not OK', [2] := 'EStop high', [3] := 'Guard doors open', [4] := 'Reject bin missing', [5] := 'No EIP connection to barcode scanner', [6] := 'No EIP connection to CTS1', [7] := 'No EIP connection to CTS2', [8] := 'No EIP connection to Robot', [9] := 'EStop Safety Block faulted', [10] := 'Barcode scanner fault', [11] := 'CTS1 fault', [12] := 'CTS2 fault', [13] := 'Robot fault', [14] := 'Robot gripper in unknown state', [15] := 'Conveyor alarm high', [16] := 'Cylinder 1 fault', [17] := 'Cylinder 2 fault', [18] := '24V DC not OK', [19] := 'Check conveyor cleat sensor', [32] := '3 in a row fault', [33] := '5 in an hour fault', [34] := '10 in a shift fault', [42] := 'Homing cycle overtime', [43] := 'Fail chute failed to register unit (Homing Seq)', [44] := 'Fail chute failed to register unit (Auto Seq)', [45] := 'Cylinder 1 down timeout', [46] := 'Cylinder 2 down timeout', [47] := 'Cylinder 1 up timeout', [48] := 'Cylinder 2 up timeout', [64] := 'Cycle stop requested', [65] := 'Cycle pause requested', [66] := 'Step mode active', [67] := 'Dry cycle active', [68] := 'MES bypass active', [74] := 'Main sequence stuck on step$0D$0A', [75] := 'Homing sequence stuck on step$0D$0A', [76] := 'CTS1 sequence stuck on step 9000', [77] := 'CTS2 sequence stuck on step 9000', [78] := 'Conveyor sequence stuck on step 9000', [79] := 'Main sequence stuck on step$0D$0A', [80] := 'Homing sequence stuck on step$0D$0A', [81] := 'CTS1 sequence stuck on step ', [82] := 'CTS2 sequence stuck on step ', [83] := 'Conveyor sequence stuck on step ', [84] := 'CTS1 test requested but interlock not met', [85] := 'CTS2 test requested but interlock not met', [86] := 'CTS1 not ready', [87] := 'CTS2 not ready', [88] := 'Robot movement requested but interlock not met', [89] := 'Conveyor movement requested but interlock not met', [90] := 'Nest 1 movement requested but interlock not met', [91] := 'Nest 2 movement requested but interlock not met', [94] := 'Fail bin full, please empty');
   FFLU_CTS1Leak : CONTROL := (LEN := 10, POS := 10, DN := 1);
   FFLU_CTS1Vol : CONTROL := (LEN := 10, POS := 10, DN := 1);
   FFLU_CTS2Leak : CONTROL := (LEN := 10, POS := 10, DN := 1);
   FFLU_CTS2Vol : CONTROL := (LEN := 10, POS := 10, DN := 1);
   FFLU_DUTHistory : CONTROL := (LEN := 10, DN := 1);
   FFLUDumpREAL : REAL;
   HMI_CloseDisplay : DINT := 12;
   HMI_OP220_ClearProcessFaultCounts_IND : BOOL;
   HMI_OP220_ClearProcessFaultCounts_PB : BOOL;
   HMI_TestPointer : DINT;
   HomingClearNestsBypass : BOOL := 1;
   InfeedCounter : COUNTER := (PRE := 9999999, ACC := 20);
   LastFaults : DINT[2] := ([0] := 205549);
   LastShiftNumber : DINT := 1;
   LeakTester1 : udt_OutputStructure := (REQ := 3);
   LeakTester2 : udt_OutputStructure := (REQ := 3);
   Mode_CapActuators : BOOL;
   Mode_CapCTS : BOOL;
   Mode_CapCylinders : BOOL;
   Mode_CapFail : BOOL;
   Mode_CapPass : BOOL;
   Mode_CapRobot : BOOL;
   Mode_CapShuffle : BOOL;
   Nest1Bypass : BOOL := 1;
   Nest1Cylinder : udt_OutputStructure := (BTMR.PRE := 500);
   Nest1Empty : BOOL := 1;
   Nest1Ready : BOOL;
   Nest2Bypass : BOOL := 1;
   Nest2Cylinder : udt_OutputStructure := (BTMR.PRE := 500);
   Nest2Empty : BOOL := 1;
   Nest2Ready : BOOL;
   ONS_AutoMode : BOOL := 1;
   ONS_CapActuators : BOOL;
   ONS_CapCTS : BOOL;
   ONS_CapCylinders : BOOL;
   ONS_CapFail : BOOL;
   ONS_CapPass : BOOL;
   ONS_CapRobot : BOOL;
   ONS_CapShuffle : BOOL;
   ONS_ClearWarnings : BOOL;
   ONS_CTS1ClearResultsBC : BOOL := 1;
   ONS_CTS1GetResults : BOOL;
   ONS_CTS1ResultHistory : BOOL;
   ONS_CTS2ClearResultsBC : BOOL := 1;
   ONS_CTS2GetResults : BOOL;
   ONS_CTS2ResultHistory : BOOL;
   ONS_CycleStop : BOOL;
   ONS_FailBinRemoved : BOOL;
   ONS_HMICloseDisplay : BOOL := 1;
   ONS_ManuMode : BOOL := 1;
   ONS_RobotGripper : SINT := 1;
   OP220 : udt_Mode := (PowerOn := 1, PowerOnONS := 1, AirOk := 1, UtilitiesOk := 1, EStopsOk := 1, GuardDoorsOk := 1, FaultActive := 1, WarningActive := 1, ReadyForAuto := 1, ManualMode := 1, Home := 1, MESBypass := 1, ManualMode_IND := 2, Home_IND := 2, HMIBackgroundIND := 2, Faults[0] := 205517, Faults[1] := 98304, Warnings[0] := 12582928, HomingOvertime.PRE := 120000, PowerOnTMR.PRE := 500, PowerOnTMR.ACC := 500, PowerOnTMR.EN := 1, PowerOnTMR.DN := 1, AirOKTMR.PRE := 500, AirOKTMR.ACC := 500, AirOKTMR.EN := 1, AirOKTMR.DN := 1, CycleStopOverideTMR.PRE := 3000, FaultTMR[0].TMR[0].PRE := 1, FaultTMR[0].TMR[1].PRE := 1, FaultTMR[0].TMR[2].PRE := 1, FaultTMR[0].TMR[3].PRE := 1, FaultTMR[0].TMR[4].PRE := 60000, FaultTMR[0].TMR[5].PRE := 1000, FaultTMR[0].TMR[5].ACC := 1000, FaultTMR[0].TMR[5].EN := 1, FaultTMR[0].TMR[5].DN := 1, FaultTMR[0].TMR[6].PRE := 1000, FaultTMR[0].TMR[6].ACC := 1000, FaultTMR[0].TMR[6].EN := 1, FaultTMR[0].TMR[6].DN := 1, FaultTMR[0].TMR[7].PRE := 1000, FaultTMR[0].TMR[7].ACC := 1000, FaultTMR[0].TMR[7].EN := 1, FaultTMR[0].TMR[7].DN := 1, FaultTMR[0].TMR[8].PRE := 1000, FaultTMR[0].TMR[9].PRE := 1, FaultTMR[0].TMR[10].PRE := 1, FaultTMR[0].TMR[11].PRE := 1, FaultTMR[0].TMR[12].PRE := 1, FaultTMR[0].TMR[13].PRE := 1, FaultTMR[0].TMR[14].PRE := 1, FaultTMR[0].TMR[15].PRE := 1000, FaultTMR[0].TMR[16].PRE := 1, FaultTMR[0].TMR[17].PRE := 1, FaultTMR[0].TMR[18].PRE := 1, FaultTMR[0].TMR[19].PRE := 1, FaultTMR[1].TMR[0].PRE := 1, FaultTMR[1].TMR[1].PRE := 1, FaultTMR[1].TMR[2].PRE := 1,
        FaultTMR[1].TMR[10].PRE := 1, FaultTMR[1].TMR[11].PRE := 1, FaultTMR[1].TMR[12].PRE := 1, FaultTMR[1].TMR[13].PRE := 1, FaultTMR[1].TMR[14].PRE := 1, FaultTMR[1].TMR[15].PRE := 1, FaultTMR[1].TMR[16].PRE := 1, FaultTMR[1].TMR[17].PRE := 1, FaultTMR[1].TMR[18].PRE := 1, FaultTMR[1].TMR[19].PRE := 1, FaultTMR[1].TMR[20].PRE := 1, WarningTMR[0].TMR[0].PRE := 1, WarningTMR[0].TMR[1].PRE := 1, WarningTMR[0].TMR[2].PRE := 1, WarningTMR[0].TMR[3].PRE := 1, WarningTMR[0].TMR[4].PRE := 1, WarningTMR[0].TMR[4].ACC := 1, WarningTMR[0].TMR[4].EN := 1, WarningTMR[0].TMR[4].DN := 1, WarningTMR[0].TMR[10].PRE := 1, WarningTMR[0].TMR[11].PRE := 1, WarningTMR[0].TMR[12].PRE := 1, WarningTMR[0].TMR[13].PRE := 1, WarningTMR[0].TMR[14].PRE := 1, WarningTMR[0].TMR[20].PRE := 2000, WarningTMR[0].TMR[21].PRE := 2000, WarningTMR[0].TMR[22].PRE := 30000, WarningTMR[0].TMR[22].ACC := 30000, WarningTMR[0].TMR[22].EN := 1, WarningTMR[0].TMR[22].DN := 1, WarningTMR[0].TMR[23].PRE := 30000, WarningTMR[0].TMR[23].ACC := 30000, WarningTMR[0].TMR[23].EN := 1, WarningTMR[0].TMR[23].DN := 1, WarningTMR[0].TMR[24].PRE := 5000, WarningTMR[0].TMR[25].PRE := 1000, WarningTMR[0].TMR[26].PRE := 1000, WarningTMR[0].TMR[27].PRE := 1000, WarningTMR[0].TMR[30].PRE := 1);
   OP220_Disable3510 : BOOL;
   OP220_Fault_Counter : COUNTER := (PRE := 9999999, ACC := 67);
   OP220_Fault_Counter_ONS : BOOL := 1;
   OP220_Fault_Number : DINT;
   OP220_Fault_Reset_ONS : BOOL;
   OP220_FaultCounter_Reset_ONS : BOOL;
   OP220_HomeONS : BOOL;
   OP220_HomingSeq : udt_SequenceStructure_X64 := (CycleDone := 1, CurrentStep := 9000, NextStep := 9000, ONS := -32768, StepHistory[0] := 1140, StepHistory[1] := 9000, StepHistory[2] := 1000, StepHistory[3] := 1020, StepHistory[4] := 1030, StepHistory[5] := 1140, StepHistory[6] := 9000, StepHistory[7] := 1000, StepHistory[8] := 1020, StepHistory[9] := 1030, StepHistory[10] := 1120, StepHistory[11] := 1140, StepHistory[12] := 9000, StepHistory[13] := 1000, StepHistory[14] := 1010, StepHistory[15] := 1020, StepHistory[16] := 1030, StepHistory[17] := 1120, StepHistory[18] := 1140, StepHistory[19] := 9000, StepHistory[20] := 1000, StepHistory[21] := 1020, StepHistory[22] := 1030, StepHistory[23] := 1120, StepHistory[24] := 1140, StepHistory[25] := 9000, StepHistory[26] := 1000, StepHistory[27] := 1020, StepHistory[28] := 1030, StepHistory[29] := 1140, StepHistory[30] := 1160, StepHistory[31] := 9000, StepHistory[32] := 1000, StepHistory[33] := 1020, StepHistory[34] := 1030, StepHistory[35] := 1140, StepHistory[36] := 1160, StepHistory[37] := 9000, StepHistory[38] := 1000, StepHistory[39] := 1020, StepHistory[40] := 1030, StepHistory[41] := 1140, StepHistory[42] := 1160, StepHistory[43] := 9000, StepHistory[44] := 1000, StepHistory[45] := 1020, StepHistory[46] := 1030, StepHistory[47] := 1120, StepHistory[48] := 1140, StepHistory[49] := 1160, StepHistory[50] := 9000, StepHistory[51] := 1000, StepHistory[52] := 1020, StepHistory[53] := 1030, StepHistory[54] := 1120, StepHistory[55] := 1140,
        StepHistory[56] := 1160, StepHistory[57] := 9000, StepHistory[58] := 1000, StepHistory[59] := 1020, StepHistory[60] := 1030, StepHistory[61] := 1120, StepHistory[62] := 1140, StepHistory[63] := 1160, StepDescriptionPointer := 1, CurrentCycleTime := 0.032, AverageCycleTime := 0.023, CycleTimeHistory[0] := 0.041, CycleTimeHistory[1] := 0.005, CycleTimeHistory[2] := 0.004, CycleTimeHistory[3] := 0.057, CycleTimeHistory[5] := 0.048, CycleTimeHistory[7] := 0.043, CycleTimeHistory[9] := 0.032, CurrentStepCycleTime := 0.028, StepTimeHistory[0] := 0.026, StepTimeHistory[1] := 0.026, StepTimeHistory[2] := 0.026, StepTimeHistory[3] := 0.026, StepTimeHistory[4] := 0.026, StepTimeHistory[5] := 0.026, StepTimeHistory[6] := 0.026, StepTimeHistory[7] := 0.026, StepTimeHistory[8] := 0.026, StepTimeHistory[9] := 0.026, StepTimeHistory[10] := 0.056, StepTimeHistory[11] := 0.056, StepTimeHistory[12] := 0.056, StepTimeHistory[13] := 0.037, StepTimeHistory[14] := 2.088, StepTimeHistory[15] := 2.088, StepTimeHistory[16] := 2.088, StepTimeHistory[17] := 0.037, StepTimeHistory[18] := 0.037, StepTimeHistory[23] := 0.038, StepTimeHistory[24] := 0.038, StepTimeHistory[25] := 0.038, StepTimeHistory[26] := 0.038, StepTimeHistory[27] := 0.038, StepTimeHistory[28] := 0.038, StepTimeHistory[29] := 0.038, StepTimeHistory[30] := 0.038, StepTimeHistory[31] := 0.038, StepTimeHistory[32] := 0.038, StepTimeHistory[33] := 0.038, StepTimeHistory[34] := 0.038, StepTimeHistory[35] := 0.038, StepTimeHistory[36] := 0.038, StepTimeHistory[37] := 0.038, StepTimeHistory[38] := 0.038, StepTimeHistory[39] := 0.052, StepTimeHistory[40] := 0.052, StepTimeHistory[41] := 0.052, StepTimeHistory[42] := 0.052, StepTimeHistory[47] := 0.042, StepTimeHistory[48] := 0.042,
        StepTimeHistory[49] := 0.042, StepTimeHistory[54] := 0.038, StepTimeHistory[55] := 0.038, StepTimeHistory[56] := 0.038, StepTimeHistory[61] := 0.028, StepTimeHistory[62] := 0.028, StepTimeHistory[63] := 0.028, StepTimer.PRE := 999999999, CycleTimer.PRE := 999999999);
   OP220_LeakTest : udt_ProcessFault;
   OP220_PartToPartCycleTMR : TIMER := (PRE := 999999999);
   OP220_ProcessFaultsONS : DINT;
   OP220_Seq : udt_SequenceStructure_X64 := (CurrentStep := 2, ONS := 2, StepHistory[0] := 9000, StepHistory[1] := 1000, StepHistory[2] := 6050, StepHistory[3] := 9000, StepHistory[4] := 1000, StepHistory[5] := 6050, StepHistory[6] := 9000, StepHistory[7] := 1000, StepHistory[8] := 6050, StepHistory[9] := 9000, StepHistory[10] := 1000, StepHistory[11] := 6050, StepHistory[12] := 9000, StepHistory[13] := 1000, StepHistory[14] := 6050, StepHistory[15] := 9000, StepHistory[16] := 1000, StepHistory[17] := 6050, StepHistory[18] := 9000, StepHistory[19] := 1000, StepHistory[20] := 6050, StepHistory[21] := 9000, StepHistory[22] := 1000, StepHistory[23] := 6050, StepHistory[24] := 9000, StepHistory[25] := 1000, StepHistory[26] := 6050, StepHistory[27] := 9000, StepHistory[28] := 1000, StepHistory[29] := 6050, StepHistory[30] := 9000, StepHistory[31] := 1000, StepHistory[32] := 6050, StepHistory[33] := 9000, StepHistory[34] := 1000, StepHistory[35] := 6050, StepHistory[36] := 9000, StepHistory[37] := 1000, StepHistory[38] := 6050, StepHistory[39] := 9000, StepHistory[40] := 1000, StepHistory[41] := 6050, StepHistory[42] := 9000, StepHistory[43] := 1000, StepHistory[44] := 6050, StepHistory[45] := 9000, StepHistory[46] := 1000, StepHistory[47] := 6050, StepHistory[48] := 9000, StepHistory[49] := 1000, StepHistory[50] := 6050, StepHistory[51] := 9000, StepHistory[52] := 1000, StepHistory[53] := 6050, StepHistory[54] := 9000, StepHistory[55] := 1000, StepHistory[56] := 6050, StepHistory[57] := 9000,
        StepHistory[58] := 1000, StepHistory[59] := 6050, StepHistory[60] := 9000, StepHistory[61] := 1000, StepHistory[62] := 6050, StepHistory[63] := 9000, StepDescriptionPointer := 1, CurrentCycleTime := 0.001, AverageCycleTime := 0.0685, PreviousCycleTime := 0.002, CycleTimeHistory[0] := 0.002, CycleTimeHistory[1] := 0.002, CycleTimeHistory[2] := 0.001, CycleTimeHistory[3] := 0.001, CycleTimeHistory[4] := 0.001, CycleTimeHistory[5] := 0.002, CycleTimeHistory[6] := 0.002, CycleTimeHistory[7] := 0.671, CycleTimeHistory[8] := 0.002, CycleTimeHistory[9] := 0.001, CurrentStepCycleTime := 0.669, StepTimeHistory[0] := 0.217, StepTimeHistory[1] := 0.217, StepTimeHistory[2] := 0.217, StepTimeHistory[3] := 0.217, StepTimeHistory[4] := 0.217, StepTimeHistory[5] := 0.217, StepTimeHistory[6] := 0.217, StepTimeHistory[7] := 0.217, StepTimeHistory[8] := 0.217, StepTimeHistory[9] := 0.217, StepTimeHistory[10] := 0.217, StepTimeHistory[11] := 0.217, StepTimeHistory[12] := 0.217, StepTimeHistory[13] := 0.217, StepTimeHistory[14] := 0.217, StepTimeHistory[15] := 0.217, StepTimeHistory[16] := 0.217, StepTimeHistory[17] := 0.217, StepTimeHistory[18] := 0.217, StepTimeHistory[19] := 0.217, StepTimeHistory[20] := 0.217, StepTimeHistory[21] := 0.217, StepTimeHistory[22] := 0.217, StepTimeHistory[23] := 0.217, StepTimeHistory[24] := 0.217, StepTimeHistory[25] := 0.217, StepTimeHistory[26] := 0.217, StepTimeHistory[27] := 0.217, StepTimeHistory[28] := 0.217, StepTimeHistory[29] := 0.217, StepTimeHistory[30] := 0.217, StepTimeHistory[31] := 0.217, StepTimeHistory[32] := 0.217, StepTimeHistory[33] := 0.217, StepTimeHistory[34] := 0.217, StepTimeHistory[35] := 0.217, StepTimeHistory[36] := 0.217, StepTimeHistory[37] := 0.217, StepTimeHistory[38] := 0.217,
        StepTimeHistory[39] := 0.217, StepTimeHistory[40] := 0.217, StepTimeHistory[41] := 0.217, StepTimeHistory[42] := 0.217, StepTimeHistory[43] := 0.217, StepTimeHistory[44] := 0.217, StepTimeHistory[45] := 0.217, StepTimeHistory[46] := 0.217, StepTimeHistory[47] := 0.217, StepTimeHistory[48] := 0.217, StepTimeHistory[49] := 0.217, StepTimeHistory[50] := 0.217, StepTimeHistory[51] := 0.217, StepTimeHistory[52] := 0.217, StepTimeHistory[53] := 0.217, StepTimeHistory[54] := 0.217, StepTimeHistory[55] := 0.669, StepTimeHistory[56] := 0.669, StepTimeHistory[57] := 0.669, StepTimeHistory[58] := 0.669, StepTimeHistory[59] := 0.669, StepTimeHistory[60] := 0.669, StepTimeHistory[61] := 0.669, StepTimeHistory[62] := 0.669, StepTimeHistory[63] := 0.669, StepTimer.PRE := 999999999, CycleTimer.PRE := 999999999);
   OutfeedCounter : COUNTER := (PRE := 9999999, ACC := 26195);
   ResetFeedCounters : BOOL;
   RFID_Comp : AOI_RFIDCompare;
   RFID_DiagData : DINT[4];
   RFID_EntryStatus : DINT;
   RFID_ExpectedFixtureVal : SINT[5,12] := ([1,0] := 26, [1,1] := 6, [1,2] := 2, [1,3] := 26, [1,5] := 7, [1,6] := 4, [1,7] := 1, [1,8] := 3, [1,10] := 1, [1,11] := 1, [2,0] := 26, [2,1] := 6, [2,2] := 2, [2,3] := 26, [2,5] := 7, [2,6] := 4, [2,7] := 1, [2,8] := 4, [2,10] := 2, [2,11] := 2);
   RFID_LoadingNestDiagData : DINT[4];
   RFID_LoadingNestReceiveBuffer : SINT[8000];
   RFID_LoadingNestSendBuffer : SINT[8000];
   RFID_PortOffset : DINT;
   RFID_ReceiveBuffer : SINT[8000];
   RFID_RWHAllPort : RWH_CMD := (isiModuleID := 13, isiFunctionID := 4, iiRdWrLength := 40);
   RFID_RWHLoadingNest : RWH_CMD := (isiModuleID := 13, isiFunctionID := 4, iiRdWrLength := 40);
   RFID_SendBuffer : SINT[8000];
   RFID_TagStatus : BOOL[32];
   RFIDLoadingNestScanner : udt_OutputStructure;
   RFIDScanner : udt_OutputStructure := (REQ := 1);
   Robot : udt_OutputStructure := (IL := 1, BC := 1, REQ := 1);
   RobotGripper : udt_OutputStructure := (IL := 1, BTMR.PRE := 2000);
   RobotInputs : udt_EpsonInputs := (ib_Ready := 1, ib_MotorsOn := 1, ib_InPos := 1, ib_GripOpen := 1, iB_SpeedEcho := 10, iW_PositionEcho := 1, iR_X := 149.65157, iR_Y := 115.6004, iR_Z := -29.66788, iR_U := 57.989914);
   RobotOutputs : udt_EpsonOutputs := (ob_SpeedOverride := 1, oB_SpeedPerc := 10, oW_TargetPosition := 1, oR_X := 191.0, oR_Y := -84.0, oR_Z := -52.0, oR_U := -270.0);
   ShiftTimes : SINT[24] := ([0] := 7, [1] := 15, [2] := 23, [3] := -1, [4] := -1, [5] := -1, [6] := -1, [7] := -1, [8] := -1, [9] := -1, [10] := -1, [11] := -1, [12] := -1, [13] := -1, [14] := -1, [15] := -1, [16] := -1, [17] := -1, [18] := -1, [19] := -1, [20] := -1, [21] := -1, [22] := -1, [23] := -1);
   TempConsumedFromPLC : BOOL;
   TempStrBuff : STRING[10] := ([0] := '9000', [1] := '/', [2] := '0', [3] := ')');
   TON_CapActuatorsDelay : TIMER := (PRE := 5000);
   TON_CapActuatorsDelay2 : TIMER := (PRE := 100);
   TON_CapCTSDelay : TIMER := (PRE := 2000);
   TON_CapCTSDelay2 : TIMER := (PRE := 2000);
   TON_CapCylindersDelay : TIMER := (PRE := 5500);
   TON_CapShuffleCTS1Delay : TIMER := (PRE := 5000);
   TON_CapShuffleCTS2Delay : TIMER := (PRE := 5000);
   TON_ConveyorCleatTimeout : TIMER := (PRE := 5000);
   TON_ConvUnloadDelay : TIMER := (PRE := 300, ACC := 300, EN := 1, DN := 1);
   TON_CTS1GetResultRetry : TIMER := (PRE := 1000);
   TON_CTS1GetResultTimeout : TIMER := (PRE := 1000);
   TON_CTS1NotGettingResultsTimeout : TIMER := (PRE := 1000);
   TON_CTS1Trigger0 : TIMER := (PRE := 200);
   TON_CTS1Trigger1 : TIMER := (PRE := 200);
   TON_CTS1Trigger2 : TIMER := (PRE := 200);
   TON_CTS2GetResultRetry : TIMER := (PRE := 1000);
   TON_CTS2GetResultTimeout : TIMER := (PRE := 1000);
   TON_CTS2NotGettingResultsTimeout : TIMER := (PRE := 1000);
   TON_CTS2Trigger0 : TIMER := (PRE := 200);
   TON_CTS2Trigger1 : TIMER := (PRE := 200);
   TON_CTS2Trigger2 : TIMER := (PRE := 1000);
   TON_Cylinder1DownTimeout : TIMER := (PRE := 5000);
   TON_Cylinder1UpTimeout : TIMER := (PRE := 5000);
   TON_Cylinder2DownTimeout : TIMER := (PRE := 5000);
   TON_Cylinder2UpTimeout : TIMER := (PRE := 5000);
   TON_FailChute : TIMER[10] := ([0].PRE := 1000, [1].PRE := 1000, [2].PRE := 1000, [3].PRE := 1000);
   TON_HMICloseDisplayDelay : TIMER := (PRE := 500);
   TON_Nest1CylinderTimer : TIMER := (PRE := 5000);
   TON_Nest1DryCycleDryTest : TIMER := (PRE := 5000);
   TON_Nest2CylinderTimer : TIMER := (PRE := 5000);
   TON_Nest2DryCycleDryTest : TIMER := (PRE := 5000);
   TON_RobotPickupSafeDelay : TIMER := (PRE := 200, ACC := 500, EN := 1, DN := 1);
   TON_RobotReqRetry : TIMER := (PRE := 1000);
   TON_RobotReqTimeout : TIMER := (PRE := 1000);
END_VAR

ROUTINE AManualDebug   (* ladder *)
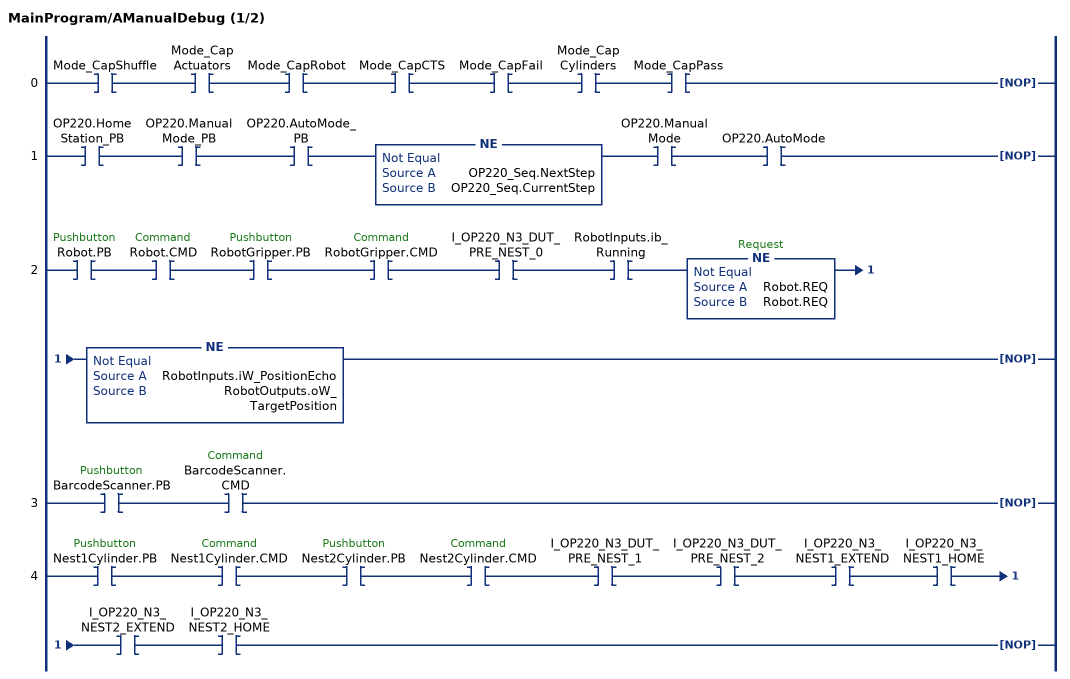
   [picture p27: MainProgram/AManualDebug rungs 0-4]
   0: XIC(Mode_CapShuffle)XIC(Mode_CapActuators)XIC(Mode_CapRobot)XIC(Mode_CapCTS)XIC(Mode_CapFail)XIC(Mode_CapCylinders)XIC(Mode_CapPass)NOP();
   1: XIC(OP220.HomeStation_PB)XIC(OP220.ManualMode_PB)XIC(OP220.AutoMode_PB)NE(OP220_Seq.NextStep,OP220_Seq.CurrentStep)XIC(OP220.ManualMode)XIC(OP220.AutoMode)NOP();
   2: XIC(Robot.PB)XIC(Robot.CMD)XIC(RobotGripper.PB)XIC(RobotGripper.CMD)XIC(I_OP220_N3_DUT_PRE_NEST_0)XIC(RobotInputs.ib_Running)NE(Robot.REQ,Robot.REQ)NE(RobotInputs.iW_PositionEcho,RobotOutputs.oW_TargetPosition)NOP();
   3: XIC(BarcodeScanner.PB)XIC(BarcodeScanner.CMD)NOP();
   4: XIC(Nest1Cylinder.PB)XIC(Nest1Cylinder.CMD)XIC(Nest2Cylinder.PB)XIC(Nest2Cylinder.CMD)XIC(I_OP220_N3_DUT_PRE_NEST_1)XIC(I_OP220_N3_DUT_PRE_NEST_2)XIC(I_OP220_N3_NEST1_EXTEND)XIC(I_OP220_N3_NEST1_HOME)XIC(I_OP220_N3_NEST2_EXTEND)XIC(I_OP220_N3_NEST2_HOME)NOP();
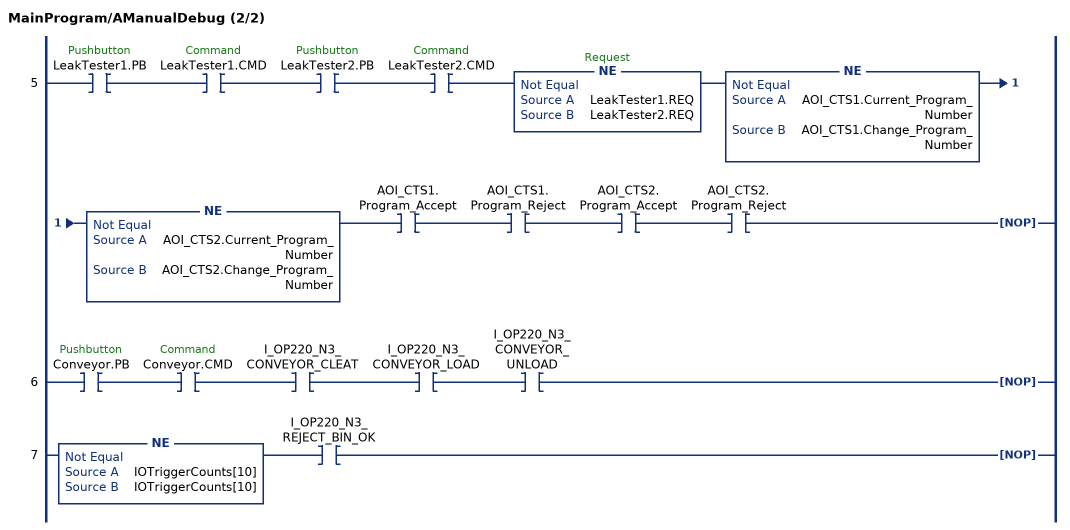
   5: XIC(LeakTester1.PB)XIC(LeakTester1.CMD)XIC(LeakTester2.PB)XIC(LeakTester2.CMD)NE(LeakTester1.REQ,LeakTester2.REQ)NE(AOI_CTS1.Current_Program_Number,AOI_CTS1.Change_Program_Number)NE(AOI_CTS2.Current_Program_Number,AOI_CTS2.Change_Program_Number)XIC(AOI_CTS1.Program_Accept)XIC(AOI_CTS1.Program_Reject)XIC(AOI_CTS2.Program_Accept)XIC(AOI_CTS2.Program_Reject)NOP();
   6: XIC(Conveyor.PB)XIC(Conveyor.CMD)XIC(I_OP220_N3_CONVEYOR_CLEAT)XIC(I_OP220_N3_CONVEYOR_LOAD)XIC(I_OP220_N3_CONVEYOR_UNLOAD)NOP();
   7: NE(IOTriggerCounts[10],IOTriggerCounts[10])XIC(I_OP220_N3_REJECT_BIN_OK)NOP();
END_ROUTINE

ROUTINE MainRoutine   (* ladder *)
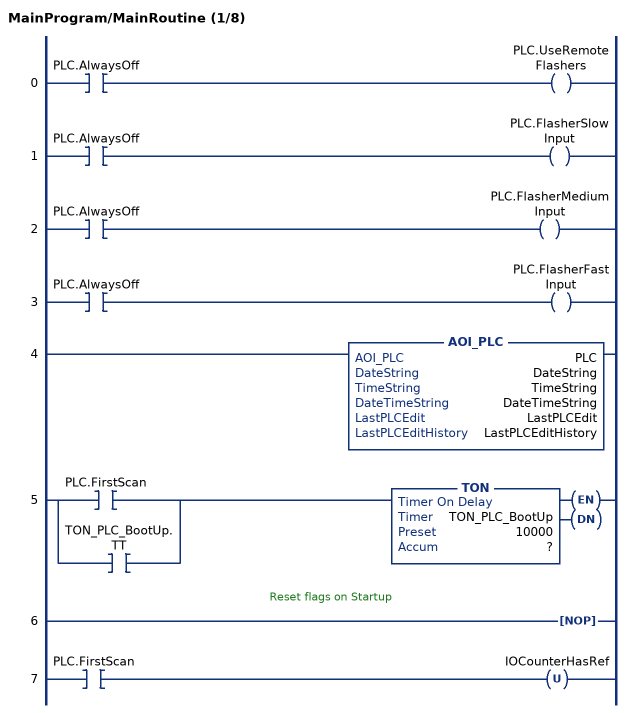
   0: XIC(PLC.AlwaysOff)OTE(PLC.UseRemoteFlashers);
   1: XIC(PLC.AlwaysOff)OTE(PLC.FlasherSlowInput);
   2: XIC(PLC.AlwaysOff)OTE(PLC.FlasherMediumInput);
   3: XIC(PLC.AlwaysOff)OTE(PLC.FlasherFastInput);
   4: AOI_PLC(PLC,DateString,TimeString,DateTimeString,LastPLCEdit,LastPLCEditHistory);
   5: [XIC(PLC.FirstScan) ,XIC(TON_PLC_BootUp.TT) ]TON(TON_PLC_BootUp,?,?);
   // Reset flags on Startup
   6: NOP();
   7: XIC(PLC.FirstScan)OTU(IOCounterHasRef);
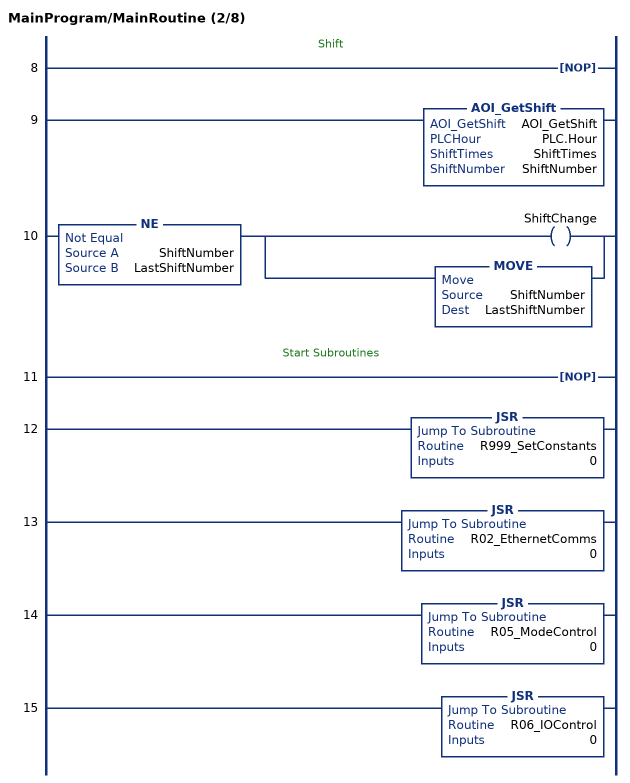
   // Shift
   8: NOP();
   9: AOI_GetShift(AOI_GetShift,PLC.Hour,ShiftTimes,ShiftNumber);
   10: NE(ShiftNumber,LastShiftNumber)[OTE(ShiftChange) ,MOVE(ShiftNumber,LastShiftNumber) ];
   // Start Subroutines
   11: NOP();
   12: JSR(R999_SetConstants,0);
   13: JSR(R02_EthernetComms,0);
   14: JSR(R05_ModeControl,0);
   15: JSR(R06_IOControl,0);
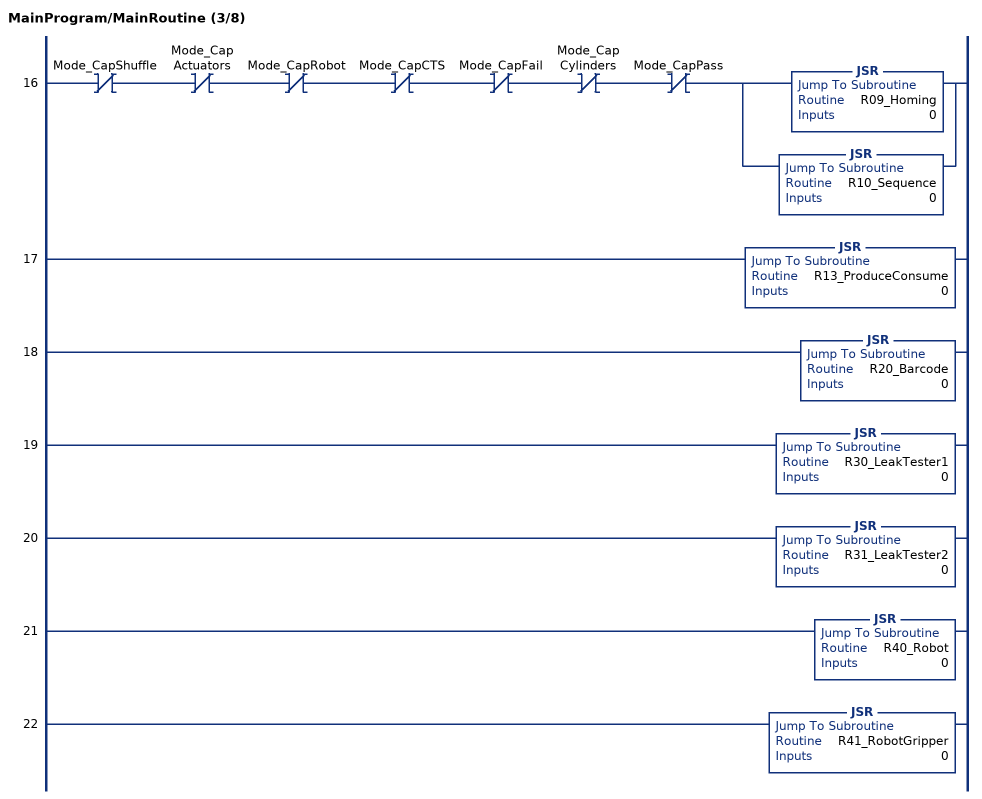
   16: XIO(Mode_CapShuffle)XIO(Mode_CapActuators)XIO(Mode_CapRobot)XIO(Mode_CapCTS)XIO(Mode_CapFail)XIO(Mode_CapCylinders)XIO(Mode_CapPass)[JSR(R09_Homing,0) ,JSR(R10_Sequence,0) ];
   17: JSR(R13_ProduceConsume,0);
   18: JSR(R20_Barcode,0);
   19: JSR(R30_LeakTester1,0);
   20: JSR(R31_LeakTester2,0);
   21: JSR(R40_Robot,0);
   22: JSR(R41_RobotGripper,0);
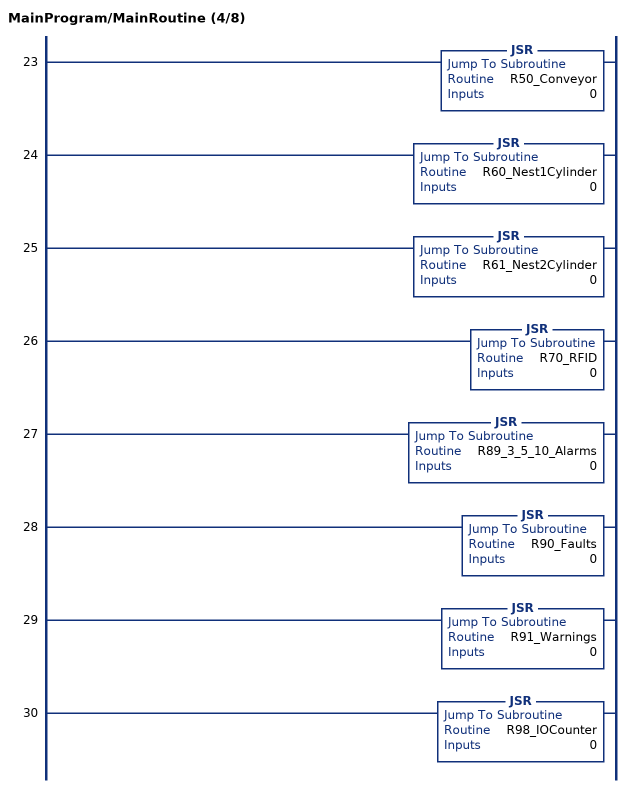
   23: JSR(R50_Conveyor,0);
   24: JSR(R60_Nest1Cylinder,0);
   25: JSR(R61_Nest2Cylinder,0);
   26: JSR(R70_RFID,0);
   27: JSR(R89_3_5_10_Alarms,0);
   28: JSR(R90_Faults,0);
   29: JSR(R91_Warnings,0);
   30: JSR(R98_IOCounter,0);
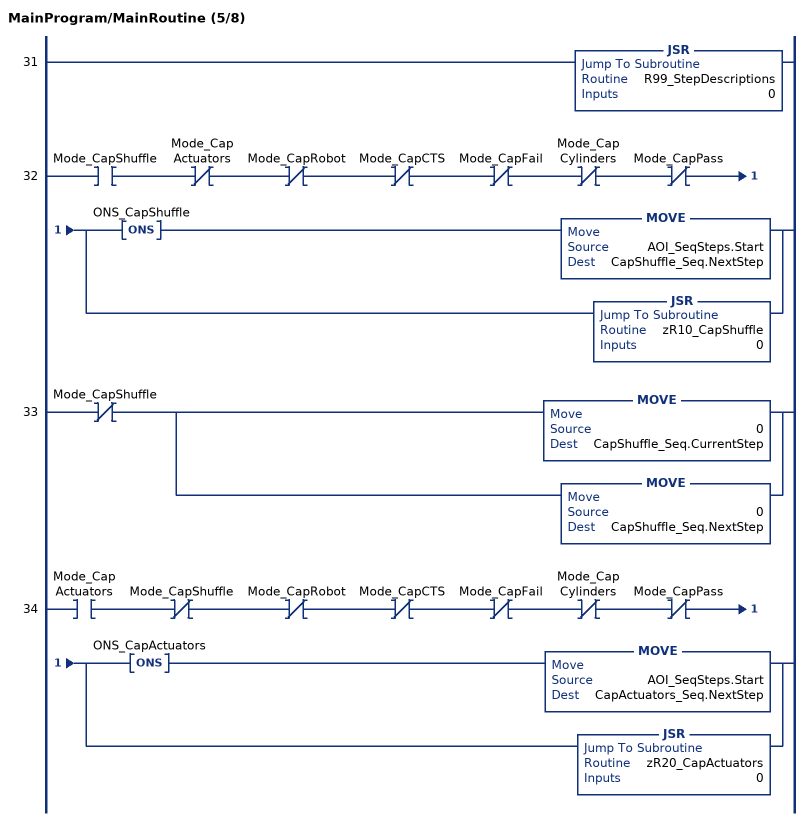
   31: JSR(R99_StepDescriptions,0);
   32: XIC(Mode_CapShuffle)XIO(Mode_CapActuators)XIO(Mode_CapRobot)XIO(Mode_CapCTS)XIO(Mode_CapFail)XIO(Mode_CapCylinders)XIO(Mode_CapPass)[ONS(ONS_CapShuffle) MOVE(AOI_SeqSteps.Start,CapShuffle_Seq.NextStep) ,JSR(zR10_CapShuffle,0) ];
   33: XIO(Mode_CapShuffle)[MOVE(0,CapShuffle_Seq.CurrentStep) ,MOVE(0,CapShuffle_Seq.NextStep) ];
   34: XIC(Mode_CapActuators)XIO(Mode_CapShuffle)XIO(Mode_CapRobot)XIO(Mode_CapCTS)XIO(Mode_CapFail)XIO(Mode_CapCylinders)XIO(Mode_CapPass)[ONS(ONS_CapActuators) MOVE(AOI_SeqSteps.Start,CapActuators_Seq.NextStep) ,JSR(zR20_CapActuators,0) ];
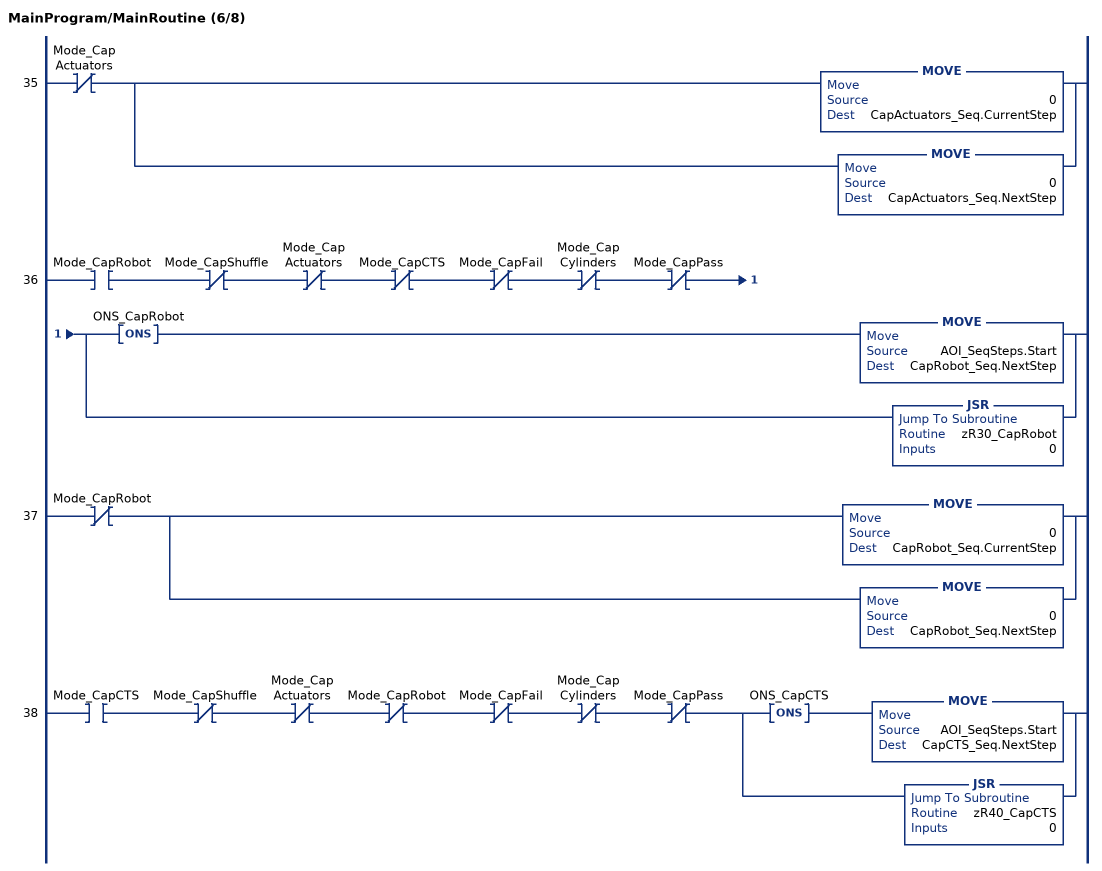
   35: XIO(Mode_CapActuators)[MOVE(0,CapActuators_Seq.CurrentStep) ,MOVE(0,CapActuators_Seq.NextStep) ];
   36: XIC(Mode_CapRobot)XIO(Mode_CapShuffle)XIO(Mode_CapActuators)XIO(Mode_CapCTS)XIO(Mode_CapFail)XIO(Mode_CapCylinders)XIO(Mode_CapPass)[ONS(ONS_CapRobot) MOVE(AOI_SeqSteps.Start,CapRobot_Seq.NextStep) ,JSR(zR30_CapRobot,0) ];
   37: XIO(Mode_CapRobot)[MOVE(0,CapRobot_Seq.CurrentStep) ,MOVE(0,CapRobot_Seq.NextStep) ];
   38: XIC(Mode_CapCTS)XIO(Mode_CapShuffle)XIO(Mode_CapActuators)XIO(Mode_CapRobot)XIO(Mode_CapFail)XIO(Mode_CapCylinders)XIO(Mode_CapPass)[ONS(ONS_CapCTS) MOVE(AOI_SeqSteps.Start,CapCTS_Seq.NextStep) ,JSR(zR40_CapCTS,0) ];
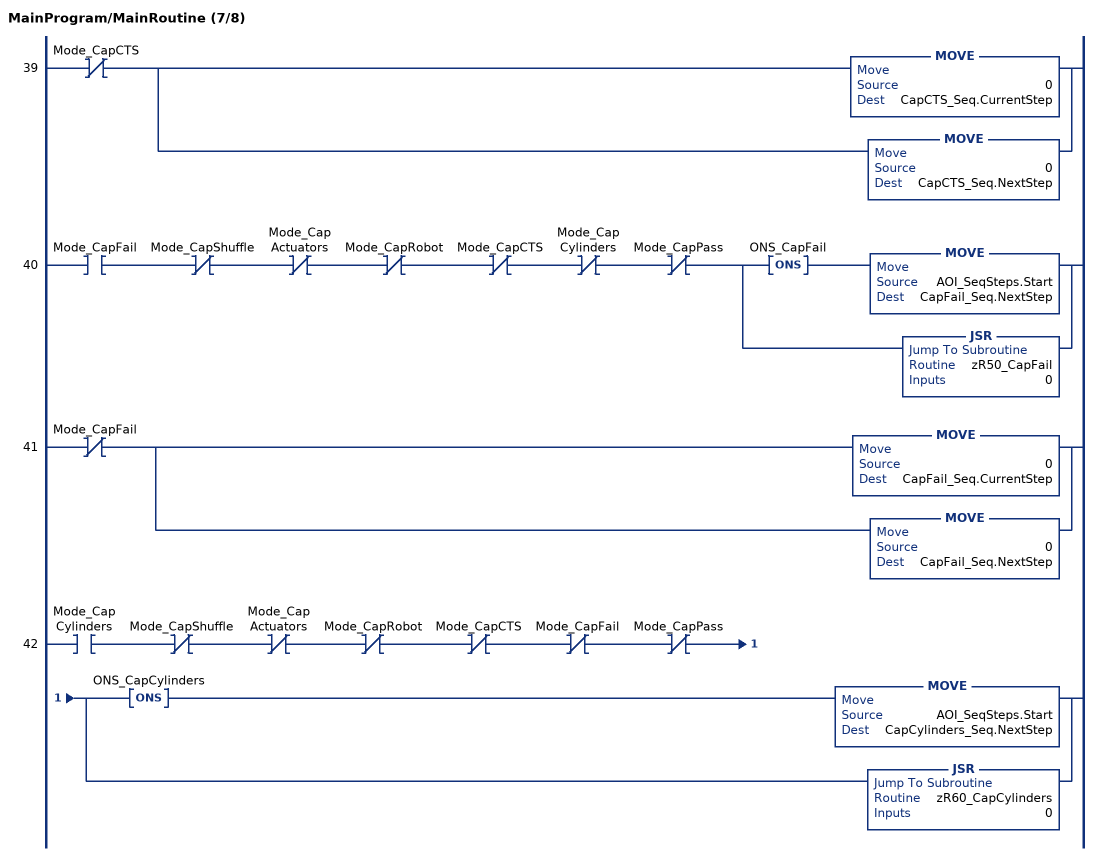
   39: XIO(Mode_CapCTS)[MOVE(0,CapCTS_Seq.CurrentStep) ,MOVE(0,CapCTS_Seq.NextStep) ];
   40: XIC(Mode_CapFail)XIO(Mode_CapShuffle)XIO(Mode_CapActuators)XIO(Mode_CapRobot)XIO(Mode_CapCTS)XIO(Mode_CapCylinders)XIO(Mode_CapPass)[ONS(ONS_CapFail) MOVE(AOI_SeqSteps.Start,CapFail_Seq.NextStep) ,JSR(zR50_CapFail,0) ];
   41: XIO(Mode_CapFail)[MOVE(0,CapFail_Seq.CurrentStep) ,MOVE(0,CapFail_Seq.NextStep) ];
   42: XIC(Mode_CapCylinders)XIO(Mode_CapShuffle)XIO(Mode_CapActuators)XIO(Mode_CapRobot)XIO(Mode_CapCTS)XIO(Mode_CapFail)XIO(Mode_CapPass)[ONS(ONS_CapCylinders) MOVE(AOI_SeqSteps.Start,CapCylinders_Seq.NextStep) ,JSR(zR60_CapCylinders,0) ];
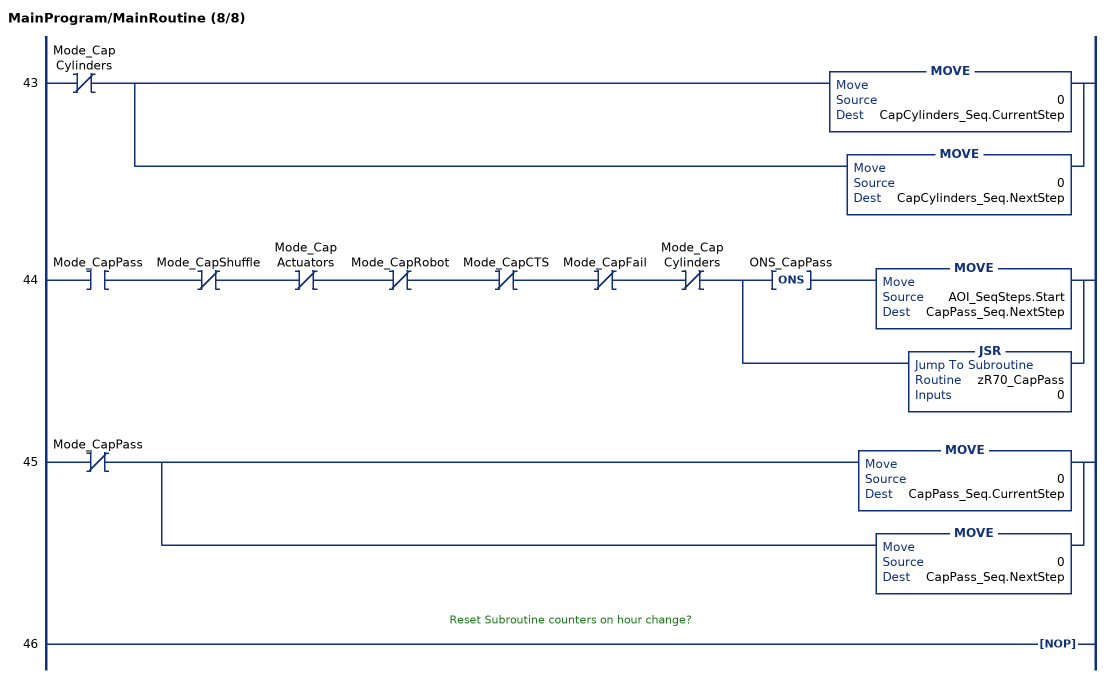
   43: XIO(Mode_CapCylinders)[MOVE(0,CapCylinders_Seq.CurrentStep) ,MOVE(0,CapCylinders_Seq.NextStep) ];
   44: XIC(Mode_CapPass)XIO(Mode_CapShuffle)XIO(Mode_CapActuators)XIO(Mode_CapRobot)XIO(Mode_CapCTS)XIO(Mode_CapFail)XIO(Mode_CapCylinders)[ONS(ONS_CapPass) MOVE(AOI_SeqSteps.Start,CapPass_Seq.NextStep) ,JSR(zR70_CapPass,0) ];
   45: XIO(Mode_CapPass)[MOVE(0,CapPass_Seq.CurrentStep) ,MOVE(0,CapPass_Seq.NextStep) ];
   // Reset Subroutine counters on hour change?
   46: NOP();
END_ROUTINE

ROUTINE R02_EthernetComms   (* ladder *)
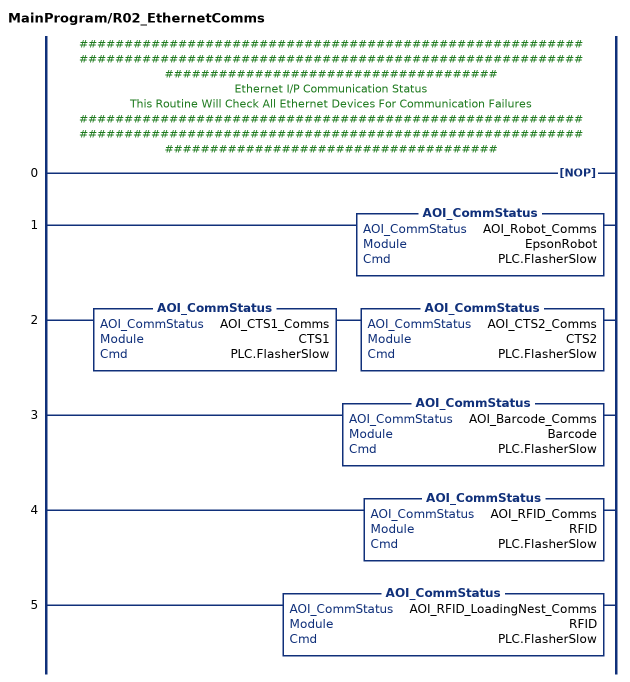
   // #####################################################################################################################################################
   // Ethernet I/P Communication Status
   // This Routine Will Check All Ethernet Devices For Communication Failures
   // #####################################################################################################################################################
   0: NOP();
   1: AOI_CommStatus(AOI_Robot_Comms,EpsonRobot,PLC.FlasherSlow);
   2: AOI_CommStatus(AOI_CTS1_Comms,CTS1,PLC.FlasherSlow)AOI_CommStatus(AOI_CTS2_Comms,CTS2,PLC.FlasherSlow);
   3: AOI_CommStatus(AOI_Barcode_Comms,Barcode,PLC.FlasherSlow);
   4: AOI_CommStatus(AOI_RFID_Comms,RFID,PLC.FlasherSlow);
   5: AOI_CommStatus(AOI_RFID_LoadingNest_Comms,RFID,PLC.FlasherSlow);
END_ROUTINE
